(* IEC 61131-3 sources: STVM/tests/functional, 4 files *)

(* ---- io_test.st ---- *)
(*
 * ============================================================================
 * STVM IO 功能综合测试 v3
 * 覆盖: 数字IO / 模拟IO / 安全输出 / 信号缩放 / PID
 * 运行: stvm tests/functional/io_test.st -I
 * ============================================================================
 *)

PROGRAM IOFunctionalTest
VAR_EXTERNAL
    button  AT %IX0.0 : BOOL;
    led     AT %QX0.0 : BOOL;
    adc_raw AT %IW0   : INT;
    pwm_out AT %QW0   : INT;
END_VAR
VAR
    raw_value   : INT;
    scaled_temp : REAL;
    error_flag  : BOOL;
    io_count    : INT;
    setpoint    : REAL;
    process_val : REAL;
    pid_output  : REAL;
    kp          : REAL;
    ki          : REAL;
    kd          : REAL;
    error_val   : REAL;
    integral    : REAL;
    derivative  : REAL;
    last_error  : REAL;
END_VAR

    PRINT('');
    PRINT('========================================');
    PRINT('  STVM IO 功能综合测试');
    PRINT('========================================');

    (* 数字 IO *)
    PRINT('--- 数字 IO ---');
    PRINT('DI button: %d', button);
    led := button;
    PRINT('DO led: %d', led);

    (* 模拟 IO *)
    PRINT('--- 模拟 IO ---');
    PRINT('AI raw: %d', adc_raw);
    pwm_out := 500;
    PRINT('AO pwm: %d', pwm_out);

    (* 信号缩放 *)
    PRINT('--- 缩放 ---');
    raw_value := adc_raw;
    scaled_temp := raw_value * 0.1;
    PRINT('Scaled: %f', scaled_temp);

    (* IO 安全检查 *)
    PRINT('--- 安全 ---');
    error_flag := FALSE;
    IF adc_raw < 0 THEN
        error_flag := TRUE;
    END_IF;
    IF error_flag THEN
        led := FALSE;
        pwm_out := 0;
        PRINT('SAFE: output disabled');
    END_IF;

    (* PID 演示 *)
    PRINT('--- PID ---');
    kp := 1.5;
    ki := 1.0;
    kd := 0.5;
    setpoint := 25.0;
    process_val := scaled_temp;
    error_val := setpoint - process_val;
    integral := integral + error_val * 0.1;
    derivative := (error_val - last_error) / 0.1;
    last_error := error_val;
    pid_output := kp * error_val + ki * integral + kd * derivative;
    PRINT('PID: SP=%f PV=%f OUT=%f', setpoint, process_val, pid_output);

    (* 周期计数器 *)
    io_count := io_count + 1;
    PRINT('IO cycle: %d', io_count);

    PRINT('========================================');
    PRINT('  IO 测试完成');
    PRINT('========================================');
END_PROGRAM

(* ---- reactor_2oo4_test.st ---- *)
(*
 * ============================================================================
 * STVM 极限性能测试 - 核反应堆 2oo4 安全控制系统 [IEC 61508 SIL3]
 * ============================================================================
 *
 * 架构:
 *   - 4 通道冗余传感器 (A/B/C/D)，每组 8 个传感器
 *   - 2oo4 表决逻辑 (4 取 2 触发)
 *   - 多重质量位传播与验证
 *   - PID 控制回路 x4 (温度/压力/流量/水位)
 *   - 安全联锁矩阵 (16x16)
 *   - 启动/运行/停机/紧急状态机
 *   - 报警管理 (16 类报警, 4 级优先级)
 *   - 所有循环带 @LOOP_MAX 标注
 *
 * 规模: ~10000 行 ST 代码, ~500+ 变量, ~80+ 函数
 * ============================================================================
 *)

PROGRAM Reactor2oo4Control

(* ================================================================ *)
(* 全局配置常量 *)
(* ================================================================ *)
VAR
    (* 系统状态 *)
    SYS_IDLE        : INT := 0;
    SYS_STARTUP     : INT := 1;
    SYS_RUNNING     : INT := 2;
    SYS_SHUTDOWN    : INT := 3;
    SYS_EMERGENCY   : INT := 4;
    system_state    : INT := 0;

    (* 安全阈值 *)
    TEMP_TRIP       : REAL := 650.0;
    PRESS_TRIP      : REAL := 15.5;
    FLOW_MIN        : REAL := 100.0;
    LEVEL_MIN       : REAL := 2.0;
    LEVEL_MAX       : REAL := 8.0;

    (* 2oo4 表决配置 *)
    VOTE_THRESHOLD  : INT := 2;
    CHANNEL_FAULT   : INT := -1;
    CHANNEL_OK      : INT := 0;

    (* 全局计数器 *)
    scan_counter    : INT := 0;
    trip_counter    : INT := 0;
    alarm_counter   : INT := 0;
    fault_counter   : INT := 0;

    (* 通用临时变量 *)
    tmp_int         : INT;
    tmp_real        : REAL;
    tmp_bool        : BOOL;
    loop_idx        : INT;
    ch_idx          : INT;
    sn_idx          : INT;
END_VAR

(* ================================================================ *)
(* 通道传感器数据 (4 通道 x 8 传感器/通道 = 32 路) *)
(* ================================================================ *)

(* 通道传感器定义 (32路) *)
FUNCTION ReadChannelA_Sensor0 : QREAL
    ReadChannelA_Sensor0 := MakeQReal(25.0, 0);
END_FUNCTION

FUNCTION ValidateChannelA_Sensor0 : BOOL
VAR_INPUT
    input_val : QREAL;
    min_limit : REAL;
    max_limit : REAL;
END_VAR
    tmp_real := ToReal(input_val);
    tmp_int := GetQuality(input_val);
    tmp_bool := FALSE;
    IF tmp_int = 0 THEN
        IF tmp_real >= min_limit THEN
            IF tmp_real <= max_limit THEN
                tmp_bool := TRUE;
            END_IF;
        END_IF;
    END_IF;
    ValidateChannelA_Sensor0 := tmp_bool;
END_FUNCTION

FUNCTION ReadChannelA_Sensor1 : QREAL
    ReadChannelA_Sensor1 := MakeQReal(25.0, 0);
END_FUNCTION

FUNCTION ValidateChannelA_Sensor1 : BOOL
VAR_INPUT
    input_val : QREAL;
    min_limit : REAL;
    max_limit : REAL;
END_VAR
    tmp_real := ToReal(input_val);
    tmp_int := GetQuality(input_val);
    tmp_bool := FALSE;
    IF tmp_int = 0 THEN
        IF tmp_real >= min_limit THEN
            IF tmp_real <= max_limit THEN
                tmp_bool := TRUE;
            END_IF;
        END_IF;
    END_IF;
    ValidateChannelA_Sensor1 := tmp_bool;
END_FUNCTION

FUNCTION ReadChannelA_Sensor2 : QREAL
    ReadChannelA_Sensor2 := MakeQReal(25.0, 0);
END_FUNCTION

FUNCTION ValidateChannelA_Sensor2 : BOOL
VAR_INPUT
    input_val : QREAL;
    min_limit : REAL;
    max_limit : REAL;
END_VAR
    tmp_real := ToReal(input_val);
    tmp_int := GetQuality(input_val);
    tmp_bool := FALSE;
    IF tmp_int = 0 THEN
        IF tmp_real >= min_limit THEN
            IF tmp_real <= max_limit THEN
                tmp_bool := TRUE;
            END_IF;
        END_IF;
    END_IF;
    ValidateChannelA_Sensor2 := tmp_bool;
END_FUNCTION

FUNCTION ReadChannelA_Sensor3 : QREAL
    ReadChannelA_Sensor3 := MakeQReal(25.0, 0);
END_FUNCTION

FUNCTION ValidateChannelA_Sensor3 : BOOL
VAR_INPUT
    input_val : QREAL;
    min_limit : REAL;
    max_limit : REAL;
END_VAR
    tmp_real := ToReal(input_val);
    tmp_int := GetQuality(input_val);
    tmp_bool := FALSE;
    IF tmp_int = 0 THEN
        IF tmp_real >= min_limit THEN
            IF tmp_real <= max_limit THEN
                tmp_bool := TRUE;
            END_IF;
        END_IF;
    END_IF;
    ValidateChannelA_Sensor3 := tmp_bool;
END_FUNCTION

FUNCTION ReadChannelA_Sensor4 : QREAL
    ReadChannelA_Sensor4 := MakeQReal(25.0, 0);
END_FUNCTION

FUNCTION ValidateChannelA_Sensor4 : BOOL
VAR_INPUT
    input_val : QREAL;
    min_limit : REAL;
    max_limit : REAL;
END_VAR
    tmp_real := ToReal(input_val);
    tmp_int := GetQuality(input_val);
    tmp_bool := FALSE;
    IF tmp_int = 0 THEN
        IF tmp_real >= min_limit THEN
            IF tmp_real <= max_limit THEN
                tmp_bool := TRUE;
            END_IF;
        END_IF;
    END_IF;
    ValidateChannelA_Sensor4 := tmp_bool;
END_FUNCTION

FUNCTION ReadChannelA_Sensor5 : QREAL
    ReadChannelA_Sensor5 := MakeQReal(25.0, 0);
END_FUNCTION

FUNCTION ValidateChannelA_Sensor5 : BOOL
VAR_INPUT
    input_val : QREAL;
    min_limit : REAL;
    max_limit : REAL;
END_VAR
    tmp_real := ToReal(input_val);
    tmp_int := GetQuality(input_val);
    tmp_bool := FALSE;
    IF tmp_int = 0 THEN
        IF tmp_real >= min_limit THEN
            IF tmp_real <= max_limit THEN
                tmp_bool := TRUE;
            END_IF;
        END_IF;
    END_IF;
    ValidateChannelA_Sensor5 := tmp_bool;
END_FUNCTION

FUNCTION ReadChannelA_Sensor6 : QREAL
    ReadChannelA_Sensor6 := MakeQReal(25.0, 0);
END_FUNCTION

FUNCTION ValidateChannelA_Sensor6 : BOOL
VAR_INPUT
    input_val : QREAL;
    min_limit : REAL;
    max_limit : REAL;
END_VAR
    tmp_real := ToReal(input_val);
    tmp_int := GetQuality(input_val);
    tmp_bool := FALSE;
    IF tmp_int = 0 THEN
        IF tmp_real >= min_limit THEN
            IF tmp_real <= max_limit THEN
                tmp_bool := TRUE;
            END_IF;
        END_IF;
    END_IF;
    ValidateChannelA_Sensor6 := tmp_bool;
END_FUNCTION

FUNCTION ReadChannelA_Sensor7 : QREAL
    ReadChannelA_Sensor7 := MakeQReal(25.0, 0);
END_FUNCTION

FUNCTION ValidateChannelA_Sensor7 : BOOL
VAR_INPUT
    input_val : QREAL;
    min_limit : REAL;
    max_limit : REAL;
END_VAR
    tmp_real := ToReal(input_val);
    tmp_int := GetQuality(input_val);
    tmp_bool := FALSE;
    IF tmp_int = 0 THEN
        IF tmp_real >= min_limit THEN
            IF tmp_real <= max_limit THEN
                tmp_bool := TRUE;
            END_IF;
        END_IF;
    END_IF;
    ValidateChannelA_Sensor7 := tmp_bool;
END_FUNCTION

FUNCTION ReadChannelB_Sensor0 : QREAL
    ReadChannelB_Sensor0 := MakeQReal(25.0, 0);
END_FUNCTION

FUNCTION ValidateChannelB_Sensor0 : BOOL
VAR_INPUT
    input_val : QREAL;
    min_limit : REAL;
    max_limit : REAL;
END_VAR
    tmp_real := ToReal(input_val);
    tmp_int := GetQuality(input_val);
    tmp_bool := FALSE;
    IF tmp_int = 0 THEN
        IF tmp_real >= min_limit THEN
            IF tmp_real <= max_limit THEN
                tmp_bool := TRUE;
            END_IF;
        END_IF;
    END_IF;
    ValidateChannelB_Sensor0 := tmp_bool;
END_FUNCTION

FUNCTION ReadChannelB_Sensor1 : QREAL
    ReadChannelB_Sensor1 := MakeQReal(25.0, 0);
END_FUNCTION

FUNCTION ValidateChannelB_Sensor1 : BOOL
VAR_INPUT
    input_val : QREAL;
    min_limit : REAL;
    max_limit : REAL;
END_VAR
    tmp_real := ToReal(input_val);
    tmp_int := GetQuality(input_val);
    tmp_bool := FALSE;
    IF tmp_int = 0 THEN
        IF tmp_real >= min_limit THEN
            IF tmp_real <= max_limit THEN
                tmp_bool := TRUE;
            END_IF;
        END_IF;
    END_IF;
    ValidateChannelB_Sensor1 := tmp_bool;
END_FUNCTION

FUNCTION ReadChannelB_Sensor2 : QREAL
    ReadChannelB_Sensor2 := MakeQReal(25.0, 0);
END_FUNCTION

FUNCTION ValidateChannelB_Sensor2 : BOOL
VAR_INPUT
    input_val : QREAL;
    min_limit : REAL;
    max_limit : REAL;
END_VAR
    tmp_real := ToReal(input_val);
    tmp_int := GetQuality(input_val);
    tmp_bool := FALSE;
    IF tmp_int = 0 THEN
        IF tmp_real >= min_limit THEN
            IF tmp_real <= max_limit THEN
                tmp_bool := TRUE;
            END_IF;
        END_IF;
    END_IF;
    ValidateChannelB_Sensor2 := tmp_bool;
END_FUNCTION

FUNCTION ReadChannelB_Sensor3 : QREAL
    ReadChannelB_Sensor3 := MakeQReal(25.0, 0);
END_FUNCTION

FUNCTION ValidateChannelB_Sensor3 : BOOL
VAR_INPUT
    input_val : QREAL;
    min_limit : REAL;
    max_limit : REAL;
END_VAR
    tmp_real := ToReal(input_val);
    tmp_int := GetQuality(input_val);
    tmp_bool := FALSE;
    IF tmp_int = 0 THEN
        IF tmp_real >= min_limit THEN
            IF tmp_real <= max_limit THEN
                tmp_bool := TRUE;
            END_IF;
        END_IF;
    END_IF;
    ValidateChannelB_Sensor3 := tmp_bool;
END_FUNCTION

FUNCTION ReadChannelB_Sensor4 : QREAL
    ReadChannelB_Sensor4 := MakeQReal(25.0, 0);
END_FUNCTION

FUNCTION ValidateChannelB_Sensor4 : BOOL
VAR_INPUT
    input_val : QREAL;
    min_limit : REAL;
    max_limit : REAL;
END_VAR
    tmp_real := ToReal(input_val);
    tmp_int := GetQuality(input_val);
    tmp_bool := FALSE;
    IF tmp_int = 0 THEN
        IF tmp_real >= min_limit THEN
            IF tmp_real <= max_limit THEN
                tmp_bool := TRUE;
            END_IF;
        END_IF;
    END_IF;
    ValidateChannelB_Sensor4 := tmp_bool;
END_FUNCTION

FUNCTION ReadChannelB_Sensor5 : QREAL
    ReadChannelB_Sensor5 := MakeQReal(25.0, 0);
END_FUNCTION

FUNCTION ValidateChannelB_Sensor5 : BOOL
VAR_INPUT
    input_val : QREAL;
    min_limit : REAL;
    max_limit : REAL;
END_VAR
    tmp_real := ToReal(input_val);
    tmp_int := GetQuality(input_val);
    tmp_bool := FALSE;
    IF tmp_int = 0 THEN
        IF tmp_real >= min_limit THEN
            IF tmp_real <= max_limit THEN
                tmp_bool := TRUE;
            END_IF;
        END_IF;
    END_IF;
    ValidateChannelB_Sensor5 := tmp_bool;
END_FUNCTION

FUNCTION ReadChannelB_Sensor6 : QREAL
    ReadChannelB_Sensor6 := MakeQReal(25.0, 0);
END_FUNCTION

FUNCTION ValidateChannelB_Sensor6 : BOOL
VAR_INPUT
    input_val : QREAL;
    min_limit : REAL;
    max_limit : REAL;
END_VAR
    tmp_real := ToReal(input_val);
    tmp_int := GetQuality(input_val);
    tmp_bool := FALSE;
    IF tmp_int = 0 THEN
        IF tmp_real >= min_limit THEN
            IF tmp_real <= max_limit THEN
                tmp_bool := TRUE;
            END_IF;
        END_IF;
    END_IF;
    ValidateChannelB_Sensor6 := tmp_bool;
END_FUNCTION

FUNCTION ReadChannelB_Sensor7 : QREAL
    ReadChannelB_Sensor7 := MakeQReal(25.0, 0);
END_FUNCTION

FUNCTION ValidateChannelB_Sensor7 : BOOL
VAR_INPUT
    input_val : QREAL;
    min_limit : REAL;
    max_limit : REAL;
END_VAR
    tmp_real := ToReal(input_val);
    tmp_int := GetQuality(input_val);
    tmp_bool := FALSE;
    IF tmp_int = 0 THEN
        IF tmp_real >= min_limit THEN
            IF tmp_real <= max_limit THEN
                tmp_bool := TRUE;
            END_IF;
        END_IF;
    END_IF;
    ValidateChannelB_Sensor7 := tmp_bool;
END_FUNCTION

FUNCTION ReadChannelC_Sensor0 : QREAL
    ReadChannelC_Sensor0 := MakeQReal(25.0, 0);
END_FUNCTION

FUNCTION ValidateChannelC_Sensor0 : BOOL
VAR_INPUT
    input_val : QREAL;
    min_limit : REAL;
    max_limit : REAL;
END_VAR
    tmp_real := ToReal(input_val);
    tmp_int := GetQuality(input_val);
    tmp_bool := FALSE;
    IF tmp_int = 0 THEN
        IF tmp_real >= min_limit THEN
            IF tmp_real <= max_limit THEN
                tmp_bool := TRUE;
            END_IF;
        END_IF;
    END_IF;
    ValidateChannelC_Sensor0 := tmp_bool;
END_FUNCTION

FUNCTION ReadChannelC_Sensor1 : QREAL
    ReadChannelC_Sensor1 := MakeQReal(25.0, 0);
END_FUNCTION

FUNCTION ValidateChannelC_Sensor1 : BOOL
VAR_INPUT
    input_val : QREAL;
    min_limit : REAL;
    max_limit : REAL;
END_VAR
    tmp_real := ToReal(input_val);
    tmp_int := GetQuality(input_val);
    tmp_bool := FALSE;
    IF tmp_int = 0 THEN
        IF tmp_real >= min_limit THEN
            IF tmp_real <= max_limit THEN
                tmp_bool := TRUE;
            END_IF;
        END_IF;
    END_IF;
    ValidateChannelC_Sensor1 := tmp_bool;
END_FUNCTION

FUNCTION ReadChannelC_Sensor2 : QREAL
    ReadChannelC_Sensor2 := MakeQReal(25.0, 0);
END_FUNCTION

FUNCTION ValidateChannelC_Sensor2 : BOOL
VAR_INPUT
    input_val : QREAL;
    min_limit : REAL;
    max_limit : REAL;
END_VAR
    tmp_real := ToReal(input_val);
    tmp_int := GetQuality(input_val);
    tmp_bool := FALSE;
    IF tmp_int = 0 THEN
        IF tmp_real >= min_limit THEN
            IF tmp_real <= max_limit THEN
                tmp_bool := TRUE;
            END_IF;
        END_IF;
    END_IF;
    ValidateChannelC_Sensor2 := tmp_bool;
END_FUNCTION

FUNCTION ReadChannelC_Sensor3 : QREAL
    ReadChannelC_Sensor3 := MakeQReal(25.0, 0);
END_FUNCTION

FUNCTION ValidateChannelC_Sensor3 : BOOL
VAR_INPUT
    input_val : QREAL;
    min_limit : REAL;
    max_limit : REAL;
END_VAR
    tmp_real := ToReal(input_val);
    tmp_int := GetQuality(input_val);
    tmp_bool := FALSE;
    IF tmp_int = 0 THEN
        IF tmp_real >= min_limit THEN
            IF tmp_real <= max_limit THEN
                tmp_bool := TRUE;
            END_IF;
        END_IF;
    END_IF;
    ValidateChannelC_Sensor3 := tmp_bool;
END_FUNCTION

FUNCTION ReadChannelC_Sensor4 : QREAL
    ReadChannelC_Sensor4 := MakeQReal(25.0, 0);
END_FUNCTION

FUNCTION ValidateChannelC_Sensor4 : BOOL
VAR_INPUT
    input_val : QREAL;
    min_limit : REAL;
    max_limit : REAL;
END_VAR
    tmp_real := ToReal(input_val);
    tmp_int := GetQuality(input_val);
    tmp_bool := FALSE;
    IF tmp_int = 0 THEN
        IF tmp_real >= min_limit THEN
            IF tmp_real <= max_limit THEN
                tmp_bool := TRUE;
            END_IF;
        END_IF;
    END_IF;
    ValidateChannelC_Sensor4 := tmp_bool;
END_FUNCTION

FUNCTION ReadChannelC_Sensor5 : QREAL
    ReadChannelC_Sensor5 := MakeQReal(25.0, 0);
END_FUNCTION

FUNCTION ValidateChannelC_Sensor5 : BOOL
VAR_INPUT
    input_val : QREAL;
    min_limit : REAL;
    max_limit : REAL;
END_VAR
    tmp_real := ToReal(input_val);
    tmp_int := GetQuality(input_val);
    tmp_bool := FALSE;
    IF tmp_int = 0 THEN
        IF tmp_real >= min_limit THEN
            IF tmp_real <= max_limit THEN
                tmp_bool := TRUE;
            END_IF;
        END_IF;
    END_IF;
    ValidateChannelC_Sensor5 := tmp_bool;
END_FUNCTION

FUNCTION ReadChannelC_Sensor6 : QREAL
    ReadChannelC_Sensor6 := MakeQReal(25.0, 0);
END_FUNCTION

FUNCTION ValidateChannelC_Sensor6 : BOOL
VAR_INPUT
    input_val : QREAL;
    min_limit : REAL;
    max_limit : REAL;
END_VAR
    tmp_real := ToReal(input_val);
    tmp_int := GetQuality(input_val);
    tmp_bool := FALSE;
    IF tmp_int = 0 THEN
        IF tmp_real >= min_limit THEN
            IF tmp_real <= max_limit THEN
                tmp_bool := TRUE;
            END_IF;
        END_IF;
    END_IF;
    ValidateChannelC_Sensor6 := tmp_bool;
END_FUNCTION

FUNCTION ReadChannelC_Sensor7 : QREAL
    ReadChannelC_Sensor7 := MakeQReal(25.0, 0);
END_FUNCTION

FUNCTION ValidateChannelC_Sensor7 : BOOL
VAR_INPUT
    input_val : QREAL;
    min_limit : REAL;
    max_limit : REAL;
END_VAR
    tmp_real := ToReal(input_val);
    tmp_int := GetQuality(input_val);
    tmp_bool := FALSE;
    IF tmp_int = 0 THEN
        IF tmp_real >= min_limit THEN
            IF tmp_real <= max_limit THEN
                tmp_bool := TRUE;
            END_IF;
        END_IF;
    END_IF;
    ValidateChannelC_Sensor7 := tmp_bool;
END_FUNCTION

FUNCTION ReadChannelD_Sensor0 : QREAL
    ReadChannelD_Sensor0 := MakeQReal(25.0, 0);
END_FUNCTION

FUNCTION ValidateChannelD_Sensor0 : BOOL
VAR_INPUT
    input_val : QREAL;
    min_limit : REAL;
    max_limit : REAL;
END_VAR
    tmp_real := ToReal(input_val);
    tmp_int := GetQuality(input_val);
    tmp_bool := FALSE;
    IF tmp_int = 0 THEN
        IF tmp_real >= min_limit THEN
            IF tmp_real <= max_limit THEN
                tmp_bool := TRUE;
            END_IF;
        END_IF;
    END_IF;
    ValidateChannelD_Sensor0 := tmp_bool;
END_FUNCTION

FUNCTION ReadChannelD_Sensor1 : QREAL
    ReadChannelD_Sensor1 := MakeQReal(25.0, 0);
END_FUNCTION

FUNCTION ValidateChannelD_Sensor1 : BOOL
VAR_INPUT
    input_val : QREAL;
    min_limit : REAL;
    max_limit : REAL;
END_VAR
    tmp_real := ToReal(input_val);
    tmp_int := GetQuality(input_val);
    tmp_bool := FALSE;
    IF tmp_int = 0 THEN
        IF tmp_real >= min_limit THEN
            IF tmp_real <= max_limit THEN
                tmp_bool := TRUE;
            END_IF;
        END_IF;
    END_IF;
    ValidateChannelD_Sensor1 := tmp_bool;
END_FUNCTION

FUNCTION ReadChannelD_Sensor2 : QREAL
    ReadChannelD_Sensor2 := MakeQReal(25.0, 0);
END_FUNCTION

FUNCTION ValidateChannelD_Sensor2 : BOOL
VAR_INPUT
    input_val : QREAL;
    min_limit : REAL;
    max_limit : REAL;
END_VAR
    tmp_real := ToReal(input_val);
    tmp_int := GetQuality(input_val);
    tmp_bool := FALSE;
    IF tmp_int = 0 THEN
        IF tmp_real >= min_limit THEN
            IF tmp_real <= max_limit THEN
                tmp_bool := TRUE;
            END_IF;
        END_IF;
    END_IF;
    ValidateChannelD_Sensor2 := tmp_bool;
END_FUNCTION

FUNCTION ReadChannelD_Sensor3 : QREAL
    ReadChannelD_Sensor3 := MakeQReal(25.0, 0);
END_FUNCTION

FUNCTION ValidateChannelD_Sensor3 : BOOL
VAR_INPUT
    input_val : QREAL;
    min_limit : REAL;
    max_limit : REAL;
END_VAR
    tmp_real := ToReal(input_val);
    tmp_int := GetQuality(input_val);
    tmp_bool := FALSE;
    IF tmp_int = 0 THEN
        IF tmp_real >= min_limit THEN
            IF tmp_real <= max_limit THEN
                tmp_bool := TRUE;
            END_IF;
        END_IF;
    END_IF;
    ValidateChannelD_Sensor3 := tmp_bool;
END_FUNCTION

FUNCTION ReadChannelD_Sensor4 : QREAL
    ReadChannelD_Sensor4 := MakeQReal(25.0, 0);
END_FUNCTION

FUNCTION ValidateChannelD_Sensor4 : BOOL
VAR_INPUT
    input_val : QREAL;
    min_limit : REAL;
    max_limit : REAL;
END_VAR
    tmp_real := ToReal(input_val);
    tmp_int := GetQuality(input_val);
    tmp_bool := FALSE;
    IF tmp_int = 0 THEN
        IF tmp_real >= min_limit THEN
            IF tmp_real <= max_limit THEN
                tmp_bool := TRUE;
            END_IF;
        END_IF;
    END_IF;
    ValidateChannelD_Sensor4 := tmp_bool;
END_FUNCTION

FUNCTION ReadChannelD_Sensor5 : QREAL
    ReadChannelD_Sensor5 := MakeQReal(25.0, 0);
END_FUNCTION

FUNCTION ValidateChannelD_Sensor5 : BOOL
VAR_INPUT
    input_val : QREAL;
    min_limit : REAL;
    max_limit : REAL;
END_VAR
    tmp_real := ToReal(input_val);
    tmp_int := GetQuality(input_val);
    tmp_bool := FALSE;
    IF tmp_int = 0 THEN
        IF tmp_real >= min_limit THEN
            IF tmp_real <= max_limit THEN
                tmp_bool := TRUE;
            END_IF;
        END_IF;
    END_IF;
    ValidateChannelD_Sensor5 := tmp_bool;
END_FUNCTION

FUNCTION ReadChannelD_Sensor6 : QREAL
    ReadChannelD_Sensor6 := MakeQReal(25.0, 0);
END_FUNCTION

FUNCTION ValidateChannelD_Sensor6 : BOOL
VAR_INPUT
    input_val : QREAL;
    min_limit : REAL;
    max_limit : REAL;
END_VAR
    tmp_real := ToReal(input_val);
    tmp_int := GetQuality(input_val);
    tmp_bool := FALSE;
    IF tmp_int = 0 THEN
        IF tmp_real >= min_limit THEN
            IF tmp_real <= max_limit THEN
                tmp_bool := TRUE;
            END_IF;
        END_IF;
    END_IF;
    ValidateChannelD_Sensor6 := tmp_bool;
END_FUNCTION

FUNCTION ReadChannelD_Sensor7 : QREAL
    ReadChannelD_Sensor7 := MakeQReal(25.0, 0);
END_FUNCTION

FUNCTION ValidateChannelD_Sensor7 : BOOL
VAR_INPUT
    input_val : QREAL;
    min_limit : REAL;
    max_limit : REAL;
END_VAR
    tmp_real := ToReal(input_val);
    tmp_int := GetQuality(input_val);
    tmp_bool := FALSE;
    IF tmp_int = 0 THEN
        IF tmp_real >= min_limit THEN
            IF tmp_real <= max_limit THEN
                tmp_bool := TRUE;
            END_IF;
        END_IF;
    END_IF;
    ValidateChannelD_Sensor7 := tmp_bool;
END_FUNCTION

(* ================================================================ *)
(* 2oo4 表决逻辑 *)
(* ================================================================ *)

FUNCTION Vote2oo4_Bool : BOOL
VAR_INPUT
    ch_a : BOOL;
    ch_b : BOOL;
    ch_c : BOOL;
    ch_d : BOOL;
END_VAR
    tmp_int := 0;
    IF ch_a THEN tmp_int := tmp_int + 1; END_IF;
    IF ch_b THEN tmp_int := tmp_int + 1; END_IF;
    IF ch_c THEN tmp_int := tmp_int + 1; END_IF;
    IF ch_d THEN tmp_int := tmp_int + 1; END_IF;
    Vote2oo4_Bool := (tmp_int >= VOTE_THRESHOLD);
END_FUNCTION

FUNCTION Vote2oo4_Real : REAL
VAR_INPUT
    ch_a : REAL;
    ch_b : REAL;
    ch_c : REAL;
    ch_d : REAL;
END_VAR
    tmp_real := ch_a + ch_b + ch_c + ch_d;
    Vote2oo4_Real := tmp_real / 4.0;
END_FUNCTION

FUNCTION Vote2oo4_QReal : QREAL
VAR_INPUT
    ch_a : QREAL;
    ch_b : QREAL;
    ch_c : QREAL;
    ch_d : QREAL;
END_VAR
    tmp_real := ToReal(ch_a) + ToReal(ch_b) + ToReal(ch_c) + ToReal(ch_d);
    Vote2oo4_QReal := MakeQReal(tmp_real / 4.0, 0);
END_FUNCTION

(* ================================================================ *)
(* @LOOP_MAX(10000) - 传感器组 0 2oo4 表决 *)
(* ================================================================ *)
FUNCTION SensorGroup0_Vote : QREAL
VAR
    s_a : QREAL;
    s_b : QREAL;
    s_c : QREAL;
    s_d : QREAL;
    v_a : BOOL;
    v_b : BOOL;
    v_c : BOOL;
    v_d : BOOL;
    vt : BOOL;
    result : QREAL;
END_VAR
    s_a := ReadChannelA_Sensor0();
    s_b := ReadChannelB_Sensor0();
    s_c := ReadChannelC_Sensor0();
    s_d := ReadChannelD_Sensor0();

    v_a := ValidateChannelA_Sensor0(s_a, 0.0, 1000.0);
    v_b := ValidateChannelB_Sensor0(s_b, 0.0, 1000.0);
    v_c := ValidateChannelC_Sensor0(s_c, 0.0, 1000.0);
    v_d := ValidateChannelD_Sensor0(s_d, 0.0, 1000.0);

    vt := Vote2oo4_Bool(v_a, v_b, v_c, v_d);
    IF vt THEN
        result := Vote2oo4_QReal(s_a, s_b, s_c, s_d);
    ELSE
        result := MakeQReal(0.0, 3);
    END_IF;
    SensorGroup0_Vote := result;
END_FUNCTION

(* ================================================================ *)
(* @LOOP_MAX(10000) - 传感器组 1 2oo4 表决 *)
(* ================================================================ *)
FUNCTION SensorGroup1_Vote : QREAL
VAR
    s_a : QREAL;
    s_b : QREAL;
    s_c : QREAL;
    s_d : QREAL;
    v_a : BOOL;
    v_b : BOOL;
    v_c : BOOL;
    v_d : BOOL;
    vt : BOOL;
    result : QREAL;
END_VAR
    s_a := ReadChannelA_Sensor1();
    s_b := ReadChannelB_Sensor1();
    s_c := ReadChannelC_Sensor1();
    s_d := ReadChannelD_Sensor1();

    v_a := ValidateChannelA_Sensor1(s_a, 0.0, 1000.0);
    v_b := ValidateChannelB_Sensor1(s_b, 0.0, 1000.0);
    v_c := ValidateChannelC_Sensor1(s_c, 0.0, 1000.0);
    v_d := ValidateChannelD_Sensor1(s_d, 0.0, 1000.0);

    vt := Vote2oo4_Bool(v_a, v_b, v_c, v_d);
    IF vt THEN
        result := Vote2oo4_QReal(s_a, s_b, s_c, s_d);
    ELSE
        result := MakeQReal(0.0, 3);
    END_IF;
    SensorGroup1_Vote := result;
END_FUNCTION

(* ================================================================ *)
(* @LOOP_MAX(10000) - 传感器组 2 2oo4 表决 *)
(* ================================================================ *)
FUNCTION SensorGroup2_Vote : QREAL
VAR
    s_a : QREAL;
    s_b : QREAL;
    s_c : QREAL;
    s_d : QREAL;
    v_a : BOOL;
    v_b : BOOL;
    v_c : BOOL;
    v_d : BOOL;
    vt : BOOL;
    result : QREAL;
END_VAR
    s_a := ReadChannelA_Sensor2();
    s_b := ReadChannelB_Sensor2();
    s_c := ReadChannelC_Sensor2();
    s_d := ReadChannelD_Sensor2();

    v_a := ValidateChannelA_Sensor2(s_a, 0.0, 1000.0);
    v_b := ValidateChannelB_Sensor2(s_b, 0.0, 1000.0);
    v_c := ValidateChannelC_Sensor2(s_c, 0.0, 1000.0);
    v_d := ValidateChannelD_Sensor2(s_d, 0.0, 1000.0);

    vt := Vote2oo4_Bool(v_a, v_b, v_c, v_d);
    IF vt THEN
        result := Vote2oo4_QReal(s_a, s_b, s_c, s_d);
    ELSE
        result := MakeQReal(0.0, 3);
    END_IF;
    SensorGroup2_Vote := result;
END_FUNCTION

(* ================================================================ *)
(* @LOOP_MAX(10000) - 传感器组 3 2oo4 表决 *)
(* ================================================================ *)
FUNCTION SensorGroup3_Vote : QREAL
VAR
    s_a : QREAL;
    s_b : QREAL;
    s_c : QREAL;
    s_d : QREAL;
    v_a : BOOL;
    v_b : BOOL;
    v_c : BOOL;
    v_d : BOOL;
    vt : BOOL;
    result : QREAL;
END_VAR
    s_a := ReadChannelA_Sensor3();
    s_b := ReadChannelB_Sensor3();
    s_c := ReadChannelC_Sensor3();
    s_d := ReadChannelD_Sensor3();

    v_a := ValidateChannelA_Sensor3(s_a, 0.0, 1000.0);
    v_b := ValidateChannelB_Sensor3(s_b, 0.0, 1000.0);
    v_c := ValidateChannelC_Sensor3(s_c, 0.0, 1000.0);
    v_d := ValidateChannelD_Sensor3(s_d, 0.0, 1000.0);

    vt := Vote2oo4_Bool(v_a, v_b, v_c, v_d);
    IF vt THEN
        result := Vote2oo4_QReal(s_a, s_b, s_c, s_d);
    ELSE
        result := MakeQReal(0.0, 3);
    END_IF;
    SensorGroup3_Vote := result;
END_FUNCTION

(* ================================================================ *)
(* @LOOP_MAX(10000) - 传感器组 4 2oo4 表决 *)
(* ================================================================ *)
FUNCTION SensorGroup4_Vote : QREAL
VAR
    s_a : QREAL;
    s_b : QREAL;
    s_c : QREAL;
    s_d : QREAL;
    v_a : BOOL;
    v_b : BOOL;
    v_c : BOOL;
    v_d : BOOL;
    vt : BOOL;
    result : QREAL;
END_VAR
    s_a := ReadChannelA_Sensor4();
    s_b := ReadChannelB_Sensor4();
    s_c := ReadChannelC_Sensor4();
    s_d := ReadChannelD_Sensor4();

    v_a := ValidateChannelA_Sensor4(s_a, 0.0, 1000.0);
    v_b := ValidateChannelB_Sensor4(s_b, 0.0, 1000.0);
    v_c := ValidateChannelC_Sensor4(s_c, 0.0, 1000.0);
    v_d := ValidateChannelD_Sensor4(s_d, 0.0, 1000.0);

    vt := Vote2oo4_Bool(v_a, v_b, v_c, v_d);
    IF vt THEN
        result := Vote2oo4_QReal(s_a, s_b, s_c, s_d);
    ELSE
        result := MakeQReal(0.0, 3);
    END_IF;
    SensorGroup4_Vote := result;
END_FUNCTION

(* ================================================================ *)
(* @LOOP_MAX(10000) - 传感器组 5 2oo4 表决 *)
(* ================================================================ *)
FUNCTION SensorGroup5_Vote : QREAL
VAR
    s_a : QREAL;
    s_b : QREAL;
    s_c : QREAL;
    s_d : QREAL;
    v_a : BOOL;
    v_b : BOOL;
    v_c : BOOL;
    v_d : BOOL;
    vt : BOOL;
    result : QREAL;
END_VAR
    s_a := ReadChannelA_Sensor5();
    s_b := ReadChannelB_Sensor5();
    s_c := ReadChannelC_Sensor5();
    s_d := ReadChannelD_Sensor5();

    v_a := ValidateChannelA_Sensor5(s_a, 0.0, 1000.0);
    v_b := ValidateChannelB_Sensor5(s_b, 0.0, 1000.0);
    v_c := ValidateChannelC_Sensor5(s_c, 0.0, 1000.0);
    v_d := ValidateChannelD_Sensor5(s_d, 0.0, 1000.0);

    vt := Vote2oo4_Bool(v_a, v_b, v_c, v_d);
    IF vt THEN
        result := Vote2oo4_QReal(s_a, s_b, s_c, s_d);
    ELSE
        result := MakeQReal(0.0, 3);
    END_IF;
    SensorGroup5_Vote := result;
END_FUNCTION

(* ================================================================ *)
(* @LOOP_MAX(10000) - 传感器组 6 2oo4 表决 *)
(* ================================================================ *)
FUNCTION SensorGroup6_Vote : QREAL
VAR
    s_a : QREAL;
    s_b : QREAL;
    s_c : QREAL;
    s_d : QREAL;
    v_a : BOOL;
    v_b : BOOL;
    v_c : BOOL;
    v_d : BOOL;
    vt : BOOL;
    result : QREAL;
END_VAR
    s_a := ReadChannelA_Sensor6();
    s_b := ReadChannelB_Sensor6();
    s_c := ReadChannelC_Sensor6();
    s_d := ReadChannelD_Sensor6();

    v_a := ValidateChannelA_Sensor6(s_a, 0.0, 1000.0);
    v_b := ValidateChannelB_Sensor6(s_b, 0.0, 1000.0);
    v_c := ValidateChannelC_Sensor6(s_c, 0.0, 1000.0);
    v_d := ValidateChannelD_Sensor6(s_d, 0.0, 1000.0);

    vt := Vote2oo4_Bool(v_a, v_b, v_c, v_d);
    IF vt THEN
        result := Vote2oo4_QReal(s_a, s_b, s_c, s_d);
    ELSE
        result := MakeQReal(0.0, 3);
    END_IF;
    SensorGroup6_Vote := result;
END_FUNCTION

(* ================================================================ *)
(* @LOOP_MAX(10000) - 传感器组 7 2oo4 表决 *)
(* ================================================================ *)
FUNCTION SensorGroup7_Vote : QREAL
VAR
    s_a : QREAL;
    s_b : QREAL;
    s_c : QREAL;
    s_d : QREAL;
    v_a : BOOL;
    v_b : BOOL;
    v_c : BOOL;
    v_d : BOOL;
    vt : BOOL;
    result : QREAL;
END_VAR
    s_a := ReadChannelA_Sensor7();
    s_b := ReadChannelB_Sensor7();
    s_c := ReadChannelC_Sensor7();
    s_d := ReadChannelD_Sensor7();

    v_a := ValidateChannelA_Sensor7(s_a, 0.0, 1000.0);
    v_b := ValidateChannelB_Sensor7(s_b, 0.0, 1000.0);
    v_c := ValidateChannelC_Sensor7(s_c, 0.0, 1000.0);
    v_d := ValidateChannelD_Sensor7(s_d, 0.0, 1000.0);

    vt := Vote2oo4_Bool(v_a, v_b, v_c, v_d);
    IF vt THEN
        result := Vote2oo4_QReal(s_a, s_b, s_c, s_d);
    ELSE
        result := MakeQReal(0.0, 3);
    END_IF;
    SensorGroup7_Vote := result;
END_FUNCTION

(* ================================================================ *)
(* PID 控制器 x4 *)
(* ================================================================ *)

FUNCTION PID_Temperature : REAL
VAR_INPUT
    sp : REAL;
    pv : REAL;
END_VAR
VAR
    kp_temp : REAL := 2.5;
    ki_temp : REAL := 0.8;
    kd_temp : REAL := 0.3;
    err     : REAL;
    integ   : REAL;
    deriv   : REAL;
    prev_err: REAL;
END_VAR
    err := sp - pv;
    integ := integ + err * 0.1;
    deriv := (err - prev_err) / 0.1;
    prev_err := err;
    PID_Temperature := kp_temp * err + ki_temp * integ + kd_temp * deriv;
END_FUNCTION

FUNCTION PID_Pressure : REAL
VAR_INPUT
    sp : REAL;
    pv : REAL;
END_VAR
VAR
    kp_val : REAL := 3.0;
    ki_val : REAL := 1.2;
    kd_val : REAL := 0.5;
    err     : REAL;
    integ   : REAL;
    deriv   : REAL;
    prev_err: REAL;
END_VAR
    err := sp - pv;
    integ := integ + err * 0.1;
    deriv := (err - prev_err) / 0.1;
    prev_err := err;
    PID_Pressure := kp_val * err + ki_val * integ + kd_val * deriv;
END_FUNCTION
FUNCTION PID_Flow : REAL
VAR_INPUT
    sp : REAL;
    pv : REAL;
END_VAR
VAR
    kp_val : REAL := 1.5;
    ki_val : REAL := 0.6;
    kd_val : REAL := 0.2;
    err     : REAL;
    integ   : REAL;
    deriv   : REAL;
    prev_err: REAL;
END_VAR
    err := sp - pv;
    integ := integ + err * 0.1;
    deriv := (err - prev_err) / 0.1;
    prev_err := err;
    PID_Flow := kp_val * err + ki_val * integ + kd_val * deriv;
END_FUNCTION
FUNCTION PID_Level : REAL
VAR_INPUT
    sp : REAL;
    pv : REAL;
END_VAR
VAR
    kp_val : REAL := 2.0;
    ki_val : REAL := 0.3;
    kd_val : REAL := 0.1;
    err     : REAL;
    integ   : REAL;
    deriv   : REAL;
    prev_err: REAL;
END_VAR
    err := sp - pv;
    integ := integ + err * 0.1;
    deriv := (err - prev_err) / 0.1;
    prev_err := err;
    PID_Level := kp_val * err + ki_val * integ + kd_val * deriv;
END_FUNCTION
(* ================================================================ *)
(* 安全联锁矩阵 16x16 *)
(* ================================================================ *)

FUNCTION InterlockMatrix : BOOL
VAR_INPUT
    signals : ARRAY[16] OF BOOL;
END_VAR
VAR
    row : INT;
    col : INT;
    result : BOOL;
END_VAR
    result := FALSE;
    FOR row := 0 TO 15 DO
        FOR col := 0 TO 15 DO
            IF signals[row] THEN
                IF signals[col] THEN
                    result := TRUE;
                END_IF;
            END_IF;
        END_FOR;
    END_FOR;
    InterlockMatrix := result;
END_FUNCTION

(* 联锁信号赋值函数 *)
FUNCTION Interlock_R0 : BOOL
VAR_INPUT
    signals : ARRAY[16] OF BOOL;
END_VAR
    Interlock_R0 := signals[0] AND signals[0];
END_FUNCTION
FUNCTION Interlock_R1 : BOOL
VAR_INPUT
    signals : ARRAY[16] OF BOOL;
END_VAR
    Interlock_R1 := signals[1] AND signals[0];
END_FUNCTION
FUNCTION Interlock_R2 : BOOL
VAR_INPUT
    signals : ARRAY[16] OF BOOL;
END_VAR
    Interlock_R2 := signals[2] AND signals[0];
END_FUNCTION
FUNCTION Interlock_R3 : BOOL
VAR_INPUT
    signals : ARRAY[16] OF BOOL;
END_VAR
    Interlock_R3 := signals[3] AND signals[0];
END_FUNCTION
FUNCTION Interlock_R4 : BOOL
VAR_INPUT
    signals : ARRAY[16] OF BOOL;
END_VAR
    Interlock_R4 := signals[4] AND signals[0];
END_FUNCTION
FUNCTION Interlock_R5 : BOOL
VAR_INPUT
    signals : ARRAY[16] OF BOOL;
END_VAR
    Interlock_R5 := signals[5] AND signals[0];
END_FUNCTION
FUNCTION Interlock_R6 : BOOL
VAR_INPUT
    signals : ARRAY[16] OF BOOL;
END_VAR
    Interlock_R6 := signals[6] AND signals[0];
END_FUNCTION
FUNCTION Interlock_R7 : BOOL
VAR_INPUT
    signals : ARRAY[16] OF BOOL;
END_VAR
    Interlock_R7 := signals[7] AND signals[0];
END_FUNCTION
FUNCTION Interlock_R8 : BOOL
VAR_INPUT
    signals : ARRAY[16] OF BOOL;
END_VAR
    Interlock_R8 := signals[8] AND signals[0];
END_FUNCTION
FUNCTION Interlock_R9 : BOOL
VAR_INPUT
    signals : ARRAY[16] OF BOOL;
END_VAR
    Interlock_R9 := signals[9] AND signals[0];
END_FUNCTION
FUNCTION Interlock_R10 : BOOL
VAR_INPUT
    signals : ARRAY[16] OF BOOL;
END_VAR
    Interlock_R10 := signals[10] AND signals[0];
END_FUNCTION
FUNCTION Interlock_R11 : BOOL
VAR_INPUT
    signals : ARRAY[16] OF BOOL;
END_VAR
    Interlock_R11 := signals[11] AND signals[0];
END_FUNCTION
FUNCTION Interlock_R12 : BOOL
VAR_INPUT
    signals : ARRAY[16] OF BOOL;
END_VAR
    Interlock_R12 := signals[12] AND signals[0];
END_FUNCTION
FUNCTION Interlock_R13 : BOOL
VAR_INPUT
    signals : ARRAY[16] OF BOOL;
END_VAR
    Interlock_R13 := signals[13] AND signals[0];
END_FUNCTION
FUNCTION Interlock_R14 : BOOL
VAR_INPUT
    signals : ARRAY[16] OF BOOL;
END_VAR
    Interlock_R14 := signals[14] AND signals[0];
END_FUNCTION
FUNCTION Interlock_R15 : BOOL
VAR_INPUT
    signals : ARRAY[16] OF BOOL;
END_VAR
    Interlock_R15 := signals[15] AND signals[0];
END_FUNCTION
(* ================================================================ *)
(* 报警管理系统 *)
(* ================================================================ *)

FUNCTION AlarmManager : INT
VAR_INPUT
    alarm_signals : ARRAY[16] OF BOOL;
END_VAR
VAR
    alm_idx : INT;
    active_count : INT;
END_VAR
    active_count := 0;
    FOR alm_idx := 0 TO 15 DO
        IF alarm_signals[alm_idx] THEN
            active_count := active_count + 1;
        END_IF;
    END_FOR;
    AlarmManager := active_count;
END_FUNCTION

FUNCTION Alarm_P1_A0 : BOOL
VAR_INPUT
    trigger : BOOL;
END_VAR
    alarm_counter := alarm_counter + 1;
    Alarm_P1_A0 := trigger;
END_FUNCTION
FUNCTION Alarm_P1_A1 : BOOL
VAR_INPUT
    trigger : BOOL;
END_VAR
    alarm_counter := alarm_counter + 1;
    Alarm_P1_A1 := trigger;
END_FUNCTION
FUNCTION Alarm_P1_A2 : BOOL
VAR_INPUT
    trigger : BOOL;
END_VAR
    alarm_counter := alarm_counter + 1;
    Alarm_P1_A2 := trigger;
END_FUNCTION
FUNCTION Alarm_P1_A3 : BOOL
VAR_INPUT
    trigger : BOOL;
END_VAR
    alarm_counter := alarm_counter + 1;
    Alarm_P1_A3 := trigger;
END_FUNCTION
FUNCTION Alarm_P2_A0 : BOOL
VAR_INPUT
    trigger : BOOL;
END_VAR
    alarm_counter := alarm_counter + 1;
    Alarm_P2_A0 := trigger;
END_FUNCTION
FUNCTION Alarm_P2_A1 : BOOL
VAR_INPUT
    trigger : BOOL;
END_VAR
    alarm_counter := alarm_counter + 1;
    Alarm_P2_A1 := trigger;
END_FUNCTION
FUNCTION Alarm_P2_A2 : BOOL
VAR_INPUT
    trigger : BOOL;
END_VAR
    alarm_counter := alarm_counter + 1;
    Alarm_P2_A2 := trigger;
END_FUNCTION
FUNCTION Alarm_P2_A3 : BOOL
VAR_INPUT
    trigger : BOOL;
END_VAR
    alarm_counter := alarm_counter + 1;
    Alarm_P2_A3 := trigger;
END_FUNCTION
FUNCTION Alarm_P3_A0 : BOOL
VAR_INPUT
    trigger : BOOL;
END_VAR
    alarm_counter := alarm_counter + 1;
    Alarm_P3_A0 := trigger;
END_FUNCTION
FUNCTION Alarm_P3_A1 : BOOL
VAR_INPUT
    trigger : BOOL;
END_VAR
    alarm_counter := alarm_counter + 1;
    Alarm_P3_A1 := trigger;
END_FUNCTION
FUNCTION Alarm_P3_A2 : BOOL
VAR_INPUT
    trigger : BOOL;
END_VAR
    alarm_counter := alarm_counter + 1;
    Alarm_P3_A2 := trigger;
END_FUNCTION
FUNCTION Alarm_P3_A3 : BOOL
VAR_INPUT
    trigger : BOOL;
END_VAR
    alarm_counter := alarm_counter + 1;
    Alarm_P3_A3 := trigger;
END_FUNCTION
FUNCTION Alarm_P4_A0 : BOOL
VAR_INPUT
    trigger : BOOL;
END_VAR
    alarm_counter := alarm_counter + 1;
    Alarm_P4_A0 := trigger;
END_FUNCTION
FUNCTION Alarm_P4_A1 : BOOL
VAR_INPUT
    trigger : BOOL;
END_VAR
    alarm_counter := alarm_counter + 1;
    Alarm_P4_A1 := trigger;
END_FUNCTION
FUNCTION Alarm_P4_A2 : BOOL
VAR_INPUT
    trigger : BOOL;
END_VAR
    alarm_counter := alarm_counter + 1;
    Alarm_P4_A2 := trigger;
END_FUNCTION
FUNCTION Alarm_P4_A3 : BOOL
VAR_INPUT
    trigger : BOOL;
END_VAR
    alarm_counter := alarm_counter + 1;
    Alarm_P4_A3 := trigger;
END_FUNCTION
(* ================================================================ *)
(* 反应堆状态机 *)
(* ================================================================ *)

FUNCTION StateMachine : INT
VAR_INPUT
    trip : BOOL;
END_VAR
VAR
    next_state : INT;
END_VAR
    next_state := system_state;
    IF trip THEN
        next_state := SYS_EMERGENCY;
    ELSIF system_state = SYS_IDLE THEN
        next_state := SYS_STARTUP;
    ELSIF system_state = SYS_STARTUP THEN
        next_state := SYS_RUNNING;
    ELSIF system_state = SYS_RUNNING THEN
        next_state := SYS_RUNNING;
    ELSIF system_state = SYS_EMERGENCY THEN
        next_state := SYS_SHUTDOWN;
    ELSIF system_state = SYS_SHUTDOWN THEN
        next_state := SYS_IDLE;
    END_IF;
    StateMachine := next_state;
END_FUNCTION

(* ================================================================ *)
(* 主控制周期 - 包含所有子系统 *)
(* ================================================================ *)

FUNCTION ControlCycle
VAR
    s0 : QREAL;
    s1 : QREAL;
    s2 : QREAL;
    s3 : QREAL;
    s4 : QREAL;
    s5 : QREAL;
    s6 : QREAL;
    s7 : QREAL;
    trip_cond : BOOL;
    avg_temp : REAL;
    avg_press : REAL;
    pid_temp : REAL;
    pid_press : REAL;
    pid_flow : REAL;
    pid_level : REAL;
    alm_signals : ARRAY[16] OF BOOL;
    alm_idx : INT;
    alm_cnt : INT;
END_VAR

    (* 读取所有传感器 *)
    s0 := SensorGroup0_Vote();
    s1 := SensorGroup1_Vote();
    s2 := SensorGroup2_Vote();
    s3 := SensorGroup3_Vote();
    s4 := SensorGroup4_Vote();
    s5 := SensorGroup5_Vote();
    s6 := SensorGroup6_Vote();
    s7 := SensorGroup7_Vote();

    (* 质量检查 *)
    tmp_int := GetQuality(s0);
    IF tmp_int > 1 THEN fault_counter := fault_counter + 1; END_IF;

    (* 2oo4 表决汇总 *)
    avg_temp := (ToReal(s0) + ToReal(s1) + ToReal(s2) + ToReal(s3)) / 4.0;
    avg_press := (ToReal(s4) + ToReal(s5) + ToReal(s6) + ToReal(s7)) / 4.0;

    (* PID 计算 *)
    pid_temp := PID_Temperature(500.0, avg_temp);
    pid_press := PID_Pressure(10.0, avg_press);
    pid_flow := PID_Flow(200.0, avg_temp * 0.5);
    pid_level := PID_Level(5.0, avg_press * 0.3);

    (* 跳闸判断 *)
    trip_cond := FALSE;
    IF avg_temp > TEMP_TRIP THEN trip_cond := TRUE; END_IF;
    IF avg_press > PRESS_TRIP THEN trip_cond := TRUE; END_IF;
    IF trip_cond THEN trip_counter := trip_counter + 1; END_IF;

    (* 报警更新 *)
    FOR alm_idx := 0 TO 15 DO
        alm_signals[alm_idx] := FALSE;
    END_FOR;
    IF avg_temp > TEMP_TRIP THEN alm_signals[0] := TRUE; END_IF;
    IF avg_press > PRESS_TRIP THEN alm_signals[1] := TRUE; END_IF;
    alm_cnt := AlarmManager(alm_signals);
    alarm_counter := alarm_counter + alm_cnt;

    (* 状态机 *)
    system_state := StateMachine(trip_cond);

    scan_counter := scan_counter + 1;
END_FUNCTION

(* @LOOP_MAX(100) - 校验函数 1 *)
FUNCTION Verify_Channel_1 : INT
VAR_INPUT
    value : REAL;
    limit : REAL;
END_VAR
    tmp_bool := (value <= limit);
    IF tmp_bool THEN
        Verify_Channel_1 := 0;
    ELSE
        Verify_Channel_1 := -1;
    END_IF;
END_FUNCTION

FUNCTION Scale_1 : REAL
VAR_INPUT
    raw : REAL;
END_VAR
    tmp_real := raw * 1.1;
    IF tmp_real > 10000.0 THEN
        tmp_real := 10000.0;
    END_IF;
    Scale_1 := tmp_real;
END_FUNCTION

FUNCTION LimitCheck_1 : BOOL
VAR_INPUT
    value : REAL;
    lo : REAL;
    hi : REAL;
END_VAR
    LimitCheck_1 := (value >= lo) AND (value <= hi);
END_FUNCTION

(* @LOOP_MAX(100) - 校验函数 2 *)
FUNCTION Verify_Channel_2 : INT
VAR_INPUT
    value : REAL;
    limit : REAL;
END_VAR
    tmp_bool := (value <= limit);
    IF tmp_bool THEN
        Verify_Channel_2 := 0;
    ELSE
        Verify_Channel_2 := -1;
    END_IF;
END_FUNCTION

FUNCTION Scale_2 : REAL
VAR_INPUT
    raw : REAL;
END_VAR
    tmp_real := raw * 1.2;
    IF tmp_real > 10000.0 THEN
        tmp_real := 10000.0;
    END_IF;
    Scale_2 := tmp_real;
END_FUNCTION

FUNCTION LimitCheck_2 : BOOL
VAR_INPUT
    value : REAL;
    lo : REAL;
    hi : REAL;
END_VAR
    LimitCheck_2 := (value >= lo) AND (value <= hi);
END_FUNCTION

(* @LOOP_MAX(100) - 校验函数 3 *)
FUNCTION Verify_Channel_3 : INT
VAR_INPUT
    value : REAL;
    limit : REAL;
END_VAR
    tmp_bool := (value <= limit);
    IF tmp_bool THEN
        Verify_Channel_3 := 0;
    ELSE
        Verify_Channel_3 := -1;
    END_IF;
END_FUNCTION

FUNCTION Scale_3 : REAL
VAR_INPUT
    raw : REAL;
END_VAR
    tmp_real := raw * 1.3;
    IF tmp_real > 10000.0 THEN
        tmp_real := 10000.0;
    END_IF;
    Scale_3 := tmp_real;
END_FUNCTION

FUNCTION LimitCheck_3 : BOOL
VAR_INPUT
    value : REAL;
    lo : REAL;
    hi : REAL;
END_VAR
    LimitCheck_3 := (value >= lo) AND (value <= hi);
END_FUNCTION

(* @LOOP_MAX(100) - 校验函数 4 *)
FUNCTION Verify_Channel_4 : INT
VAR_INPUT
    value : REAL;
    limit : REAL;
END_VAR
    tmp_bool := (value <= limit);
    IF tmp_bool THEN
        Verify_Channel_4 := 0;
    ELSE
        Verify_Channel_4 := -1;
    END_IF;
END_FUNCTION

FUNCTION Scale_4 : REAL
VAR_INPUT
    raw : REAL;
END_VAR
    tmp_real := raw * 1.4;
    IF tmp_real > 10000.0 THEN
        tmp_real := 10000.0;
    END_IF;
    Scale_4 := tmp_real;
END_FUNCTION

FUNCTION LimitCheck_4 : BOOL
VAR_INPUT
    value : REAL;
    lo : REAL;
    hi : REAL;
END_VAR
    LimitCheck_4 := (value >= lo) AND (value <= hi);
END_FUNCTION

(* @LOOP_MAX(100) - 校验函数 5 *)
FUNCTION Verify_Channel_5 : INT
VAR_INPUT
    value : REAL;
    limit : REAL;
END_VAR
    tmp_bool := (value <= limit);
    IF tmp_bool THEN
        Verify_Channel_5 := 0;
    ELSE
        Verify_Channel_5 := -1;
    END_IF;
END_FUNCTION

FUNCTION Scale_5 : REAL
VAR_INPUT
    raw : REAL;
END_VAR
    tmp_real := raw * 1.5;
    IF tmp_real > 10000.0 THEN
        tmp_real := 10000.0;
    END_IF;
    Scale_5 := tmp_real;
END_FUNCTION

FUNCTION LimitCheck_5 : BOOL
VAR_INPUT
    value : REAL;
    lo : REAL;
    hi : REAL;
END_VAR
    LimitCheck_5 := (value >= lo) AND (value <= hi);
END_FUNCTION

(* @LOOP_MAX(100) - 校验函数 6 *)
FUNCTION Verify_Channel_6 : INT
VAR_INPUT
    value : REAL;
    limit : REAL;
END_VAR
    tmp_bool := (value <= limit);
    IF tmp_bool THEN
        Verify_Channel_6 := 0;
    ELSE
        Verify_Channel_6 := -1;
    END_IF;
END_FUNCTION

FUNCTION Scale_6 : REAL
VAR_INPUT
    raw : REAL;
END_VAR
    tmp_real := raw * 1.6;
    IF tmp_real > 10000.0 THEN
        tmp_real := 10000.0;
    END_IF;
    Scale_6 := tmp_real;
END_FUNCTION

FUNCTION LimitCheck_6 : BOOL
VAR_INPUT
    value : REAL;
    lo : REAL;
    hi : REAL;
END_VAR
    LimitCheck_6 := (value >= lo) AND (value <= hi);
END_FUNCTION

(* @LOOP_MAX(100) - 校验函数 7 *)
FUNCTION Verify_Channel_7 : INT
VAR_INPUT
    value : REAL;
    limit : REAL;
END_VAR
    tmp_bool := (value <= limit);
    IF tmp_bool THEN
        Verify_Channel_7 := 0;
    ELSE
        Verify_Channel_7 := -1;
    END_IF;
END_FUNCTION

FUNCTION Scale_7 : REAL
VAR_INPUT
    raw : REAL;
END_VAR
    tmp_real := raw * 1.7;
    IF tmp_real > 10000.0 THEN
        tmp_real := 10000.0;
    END_IF;
    Scale_7 := tmp_real;
END_FUNCTION

FUNCTION LimitCheck_7 : BOOL
VAR_INPUT
    value : REAL;
    lo : REAL;
    hi : REAL;
END_VAR
    LimitCheck_7 := (value >= lo) AND (value <= hi);
END_FUNCTION

(* @LOOP_MAX(100) - 校验函数 8 *)
FUNCTION Verify_Channel_8 : INT
VAR_INPUT
    value : REAL;
    limit : REAL;
END_VAR
    tmp_bool := (value <= limit);
    IF tmp_bool THEN
        Verify_Channel_8 := 0;
    ELSE
        Verify_Channel_8 := -1;
    END_IF;
END_FUNCTION

FUNCTION Scale_8 : REAL
VAR_INPUT
    raw : REAL;
END_VAR
    tmp_real := raw * 1.8;
    IF tmp_real > 10000.0 THEN
        tmp_real := 10000.0;
    END_IF;
    Scale_8 := tmp_real;
END_FUNCTION

FUNCTION LimitCheck_8 : BOOL
VAR_INPUT
    value : REAL;
    lo : REAL;
    hi : REAL;
END_VAR
    LimitCheck_8 := (value >= lo) AND (value <= hi);
END_FUNCTION

(* @LOOP_MAX(100) - 校验函数 9 *)
FUNCTION Verify_Channel_9 : INT
VAR_INPUT
    value : REAL;
    limit : REAL;
END_VAR
    tmp_bool := (value <= limit);
    IF tmp_bool THEN
        Verify_Channel_9 := 0;
    ELSE
        Verify_Channel_9 := -1;
    END_IF;
END_FUNCTION

FUNCTION Scale_9 : REAL
VAR_INPUT
    raw : REAL;
END_VAR
    tmp_real := raw * 1.9;
    IF tmp_real > 10000.0 THEN
        tmp_real := 10000.0;
    END_IF;
    Scale_9 := tmp_real;
END_FUNCTION

FUNCTION LimitCheck_9 : BOOL
VAR_INPUT
    value : REAL;
    lo : REAL;
    hi : REAL;
END_VAR
    LimitCheck_9 := (value >= lo) AND (value <= hi);
END_FUNCTION

(* @LOOP_MAX(100) - 校验函数 10 *)
FUNCTION Verify_Channel_10 : INT
VAR_INPUT
    value : REAL;
    limit : REAL;
END_VAR
    tmp_bool := (value <= limit);
    IF tmp_bool THEN
        Verify_Channel_10 := 0;
    ELSE
        Verify_Channel_10 := -1;
    END_IF;
END_FUNCTION

FUNCTION Scale_10 : REAL
VAR_INPUT
    raw : REAL;
END_VAR
    tmp_real := raw * 1.10;
    IF tmp_real > 10000.0 THEN
        tmp_real := 10000.0;
    END_IF;
    Scale_10 := tmp_real;
END_FUNCTION

FUNCTION LimitCheck_10 : BOOL
VAR_INPUT
    value : REAL;
    lo : REAL;
    hi : REAL;
END_VAR
    LimitCheck_10 := (value >= lo) AND (value <= hi);
END_FUNCTION

(* @LOOP_MAX(100) - 校验函数 11 *)
FUNCTION Verify_Channel_11 : INT
VAR_INPUT
    value : REAL;
    limit : REAL;
END_VAR
    tmp_bool := (value <= limit);
    IF tmp_bool THEN
        Verify_Channel_11 := 0;
    ELSE
        Verify_Channel_11 := -1;
    END_IF;
END_FUNCTION

FUNCTION Scale_11 : REAL
VAR_INPUT
    raw : REAL;
END_VAR
    tmp_real := raw * 1.11;
    IF tmp_real > 10000.0 THEN
        tmp_real := 10000.0;
    END_IF;
    Scale_11 := tmp_real;
END_FUNCTION

FUNCTION LimitCheck_11 : BOOL
VAR_INPUT
    value : REAL;
    lo : REAL;
    hi : REAL;
END_VAR
    LimitCheck_11 := (value >= lo) AND (value <= hi);
END_FUNCTION

(* @LOOP_MAX(100) - 校验函数 12 *)
FUNCTION Verify_Channel_12 : INT
VAR_INPUT
    value : REAL;
    limit : REAL;
END_VAR
    tmp_bool := (value <= limit);
    IF tmp_bool THEN
        Verify_Channel_12 := 0;
    ELSE
        Verify_Channel_12 := -1;
    END_IF;
END_FUNCTION

FUNCTION Scale_12 : REAL
VAR_INPUT
    raw : REAL;
END_VAR
    tmp_real := raw * 1.12;
    IF tmp_real > 10000.0 THEN
        tmp_real := 10000.0;
    END_IF;
    Scale_12 := tmp_real;
END_FUNCTION

FUNCTION LimitCheck_12 : BOOL
VAR_INPUT
    value : REAL;
    lo : REAL;
    hi : REAL;
END_VAR
    LimitCheck_12 := (value >= lo) AND (value <= hi);
END_FUNCTION

(* @LOOP_MAX(100) - 校验函数 13 *)
FUNCTION Verify_Channel_13 : INT
VAR_INPUT
    value : REAL;
    limit : REAL;
END_VAR
    tmp_bool := (value <= limit);
    IF tmp_bool THEN
        Verify_Channel_13 := 0;
    ELSE
        Verify_Channel_13 := -1;
    END_IF;
END_FUNCTION

FUNCTION Scale_13 : REAL
VAR_INPUT
    raw : REAL;
END_VAR
    tmp_real := raw * 1.13;
    IF tmp_real > 10000.0 THEN
        tmp_real := 10000.0;
    END_IF;
    Scale_13 := tmp_real;
END_FUNCTION

FUNCTION LimitCheck_13 : BOOL
VAR_INPUT
    value : REAL;
    lo : REAL;
    hi : REAL;
END_VAR
    LimitCheck_13 := (value >= lo) AND (value <= hi);
END_FUNCTION

(* @LOOP_MAX(100) - 校验函数 14 *)
FUNCTION Verify_Channel_14 : INT
VAR_INPUT
    value : REAL;
    limit : REAL;
END_VAR
    tmp_bool := (value <= limit);
    IF tmp_bool THEN
        Verify_Channel_14 := 0;
    ELSE
        Verify_Channel_14 := -1;
    END_IF;
END_FUNCTION

FUNCTION Scale_14 : REAL
VAR_INPUT
    raw : REAL;
END_VAR
    tmp_real := raw * 1.14;
    IF tmp_real > 10000.0 THEN
        tmp_real := 10000.0;
    END_IF;
    Scale_14 := tmp_real;
END_FUNCTION

FUNCTION LimitCheck_14 : BOOL
VAR_INPUT
    value : REAL;
    lo : REAL;
    hi : REAL;
END_VAR
    LimitCheck_14 := (value >= lo) AND (value <= hi);
END_FUNCTION

(* @LOOP_MAX(100) - 校验函数 15 *)
FUNCTION Verify_Channel_15 : INT
VAR_INPUT
    value : REAL;
    limit : REAL;
END_VAR
    tmp_bool := (value <= limit);
    IF tmp_bool THEN
        Verify_Channel_15 := 0;
    ELSE
        Verify_Channel_15 := -1;
    END_IF;
END_FUNCTION

FUNCTION Scale_15 : REAL
VAR_INPUT
    raw : REAL;
END_VAR
    tmp_real := raw * 1.15;
    IF tmp_real > 10000.0 THEN
        tmp_real := 10000.0;
    END_IF;
    Scale_15 := tmp_real;
END_FUNCTION

FUNCTION LimitCheck_15 : BOOL
VAR_INPUT
    value : REAL;
    lo : REAL;
    hi : REAL;
END_VAR
    LimitCheck_15 := (value >= lo) AND (value <= hi);
END_FUNCTION

(* @LOOP_MAX(100) - 校验函数 16 *)
FUNCTION Verify_Channel_16 : INT
VAR_INPUT
    value : REAL;
    limit : REAL;
END_VAR
    tmp_bool := (value <= limit);
    IF tmp_bool THEN
        Verify_Channel_16 := 0;
    ELSE
        Verify_Channel_16 := -1;
    END_IF;
END_FUNCTION

FUNCTION Scale_16 : REAL
VAR_INPUT
    raw : REAL;
END_VAR
    tmp_real := raw * 1.16;
    IF tmp_real > 10000.0 THEN
        tmp_real := 10000.0;
    END_IF;
    Scale_16 := tmp_real;
END_FUNCTION

FUNCTION LimitCheck_16 : BOOL
VAR_INPUT
    value : REAL;
    lo : REAL;
    hi : REAL;
END_VAR
    LimitCheck_16 := (value >= lo) AND (value <= hi);
END_FUNCTION

(* @LOOP_MAX(100) - 校验函数 17 *)
FUNCTION Verify_Channel_17 : INT
VAR_INPUT
    value : REAL;
    limit : REAL;
END_VAR
    tmp_bool := (value <= limit);
    IF tmp_bool THEN
        Verify_Channel_17 := 0;
    ELSE
        Verify_Channel_17 := -1;
    END_IF;
END_FUNCTION

FUNCTION Scale_17 : REAL
VAR_INPUT
    raw : REAL;
END_VAR
    tmp_real := raw * 1.17;
    IF tmp_real > 10000.0 THEN
        tmp_real := 10000.0;
    END_IF;
    Scale_17 := tmp_real;
END_FUNCTION

FUNCTION LimitCheck_17 : BOOL
VAR_INPUT
    value : REAL;
    lo : REAL;
    hi : REAL;
END_VAR
    LimitCheck_17 := (value >= lo) AND (value <= hi);
END_FUNCTION

(* @LOOP_MAX(100) - 校验函数 18 *)
FUNCTION Verify_Channel_18 : INT
VAR_INPUT
    value : REAL;
    limit : REAL;
END_VAR
    tmp_bool := (value <= limit);
    IF tmp_bool THEN
        Verify_Channel_18 := 0;
    ELSE
        Verify_Channel_18 := -1;
    END_IF;
END_FUNCTION

FUNCTION Scale_18 : REAL
VAR_INPUT
    raw : REAL;
END_VAR
    tmp_real := raw * 1.18;
    IF tmp_real > 10000.0 THEN
        tmp_real := 10000.0;
    END_IF;
    Scale_18 := tmp_real;
END_FUNCTION

FUNCTION LimitCheck_18 : BOOL
VAR_INPUT
    value : REAL;
    lo : REAL;
    hi : REAL;
END_VAR
    LimitCheck_18 := (value >= lo) AND (value <= hi);
END_FUNCTION

(* @LOOP_MAX(100) - 校验函数 19 *)
FUNCTION Verify_Channel_19 : INT
VAR_INPUT
    value : REAL;
    limit : REAL;
END_VAR
    tmp_bool := (value <= limit);
    IF tmp_bool THEN
        Verify_Channel_19 := 0;
    ELSE
        Verify_Channel_19 := -1;
    END_IF;
END_FUNCTION

FUNCTION Scale_19 : REAL
VAR_INPUT
    raw : REAL;
END_VAR
    tmp_real := raw * 1.19;
    IF tmp_real > 10000.0 THEN
        tmp_real := 10000.0;
    END_IF;
    Scale_19 := tmp_real;
END_FUNCTION

FUNCTION LimitCheck_19 : BOOL
VAR_INPUT
    value : REAL;
    lo : REAL;
    hi : REAL;
END_VAR
    LimitCheck_19 := (value >= lo) AND (value <= hi);
END_FUNCTION

(* @LOOP_MAX(100) - 校验函数 20 *)
FUNCTION Verify_Channel_20 : INT
VAR_INPUT
    value : REAL;
    limit : REAL;
END_VAR
    tmp_bool := (value <= limit);
    IF tmp_bool THEN
        Verify_Channel_20 := 0;
    ELSE
        Verify_Channel_20 := -1;
    END_IF;
END_FUNCTION

FUNCTION Scale_20 : REAL
VAR_INPUT
    raw : REAL;
END_VAR
    tmp_real := raw * 1.20;
    IF tmp_real > 10000.0 THEN
        tmp_real := 10000.0;
    END_IF;
    Scale_20 := tmp_real;
END_FUNCTION

FUNCTION LimitCheck_20 : BOOL
VAR_INPUT
    value : REAL;
    lo : REAL;
    hi : REAL;
END_VAR
    LimitCheck_20 := (value >= lo) AND (value <= hi);
END_FUNCTION

(* @LOOP_MAX(100) - 校验函数 21 *)
FUNCTION Verify_Channel_21 : INT
VAR_INPUT
    value : REAL;
    limit : REAL;
END_VAR
    tmp_bool := (value <= limit);
    IF tmp_bool THEN
        Verify_Channel_21 := 0;
    ELSE
        Verify_Channel_21 := -1;
    END_IF;
END_FUNCTION

FUNCTION Scale_21 : REAL
VAR_INPUT
    raw : REAL;
END_VAR
    tmp_real := raw * 1.21;
    IF tmp_real > 10000.0 THEN
        tmp_real := 10000.0;
    END_IF;
    Scale_21 := tmp_real;
END_FUNCTION

FUNCTION LimitCheck_21 : BOOL
VAR_INPUT
    value : REAL;
    lo : REAL;
    hi : REAL;
END_VAR
    LimitCheck_21 := (value >= lo) AND (value <= hi);
END_FUNCTION

(* @LOOP_MAX(100) - 校验函数 22 *)
FUNCTION Verify_Channel_22 : INT
VAR_INPUT
    value : REAL;
    limit : REAL;
END_VAR
    tmp_bool := (value <= limit);
    IF tmp_bool THEN
        Verify_Channel_22 := 0;
    ELSE
        Verify_Channel_22 := -1;
    END_IF;
END_FUNCTION

FUNCTION Scale_22 : REAL
VAR_INPUT
    raw : REAL;
END_VAR
    tmp_real := raw * 1.22;
    IF tmp_real > 10000.0 THEN
        tmp_real := 10000.0;
    END_IF;
    Scale_22 := tmp_real;
END_FUNCTION

FUNCTION LimitCheck_22 : BOOL
VAR_INPUT
    value : REAL;
    lo : REAL;
    hi : REAL;
END_VAR
    LimitCheck_22 := (value >= lo) AND (value <= hi);
END_FUNCTION

(* @LOOP_MAX(100) - 校验函数 23 *)
FUNCTION Verify_Channel_23 : INT
VAR_INPUT
    value : REAL;
    limit : REAL;
END_VAR
    tmp_bool := (value <= limit);
    IF tmp_bool THEN
        Verify_Channel_23 := 0;
    ELSE
        Verify_Channel_23 := -1;
    END_IF;
END_FUNCTION

FUNCTION Scale_23 : REAL
VAR_INPUT
    raw : REAL;
END_VAR
    tmp_real := raw * 1.23;
    IF tmp_real > 10000.0 THEN
        tmp_real := 10000.0;
    END_IF;
    Scale_23 := tmp_real;
END_FUNCTION

FUNCTION LimitCheck_23 : BOOL
VAR_INPUT
    value : REAL;
    lo : REAL;
    hi : REAL;
END_VAR
    LimitCheck_23 := (value >= lo) AND (value <= hi);
END_FUNCTION

(* @LOOP_MAX(100) - 校验函数 24 *)
FUNCTION Verify_Channel_24 : INT
VAR_INPUT
    value : REAL;
    limit : REAL;
END_VAR
    tmp_bool := (value <= limit);
    IF tmp_bool THEN
        Verify_Channel_24 := 0;
    ELSE
        Verify_Channel_24 := -1;
    END_IF;
END_FUNCTION

FUNCTION Scale_24 : REAL
VAR_INPUT
    raw : REAL;
END_VAR
    tmp_real := raw * 1.24;
    IF tmp_real > 10000.0 THEN
        tmp_real := 10000.0;
    END_IF;
    Scale_24 := tmp_real;
END_FUNCTION

FUNCTION LimitCheck_24 : BOOL
VAR_INPUT
    value : REAL;
    lo : REAL;
    hi : REAL;
END_VAR
    LimitCheck_24 := (value >= lo) AND (value <= hi);
END_FUNCTION

(* @LOOP_MAX(100) - 校验函数 25 *)
FUNCTION Verify_Channel_25 : INT
VAR_INPUT
    value : REAL;
    limit : REAL;
END_VAR
    tmp_bool := (value <= limit);
    IF tmp_bool THEN
        Verify_Channel_25 := 0;
    ELSE
        Verify_Channel_25 := -1;
    END_IF;
END_FUNCTION

FUNCTION Scale_25 : REAL
VAR_INPUT
    raw : REAL;
END_VAR
    tmp_real := raw * 1.25;
    IF tmp_real > 10000.0 THEN
        tmp_real := 10000.0;
    END_IF;
    Scale_25 := tmp_real;
END_FUNCTION

FUNCTION LimitCheck_25 : BOOL
VAR_INPUT
    value : REAL;
    lo : REAL;
    hi : REAL;
END_VAR
    LimitCheck_25 := (value >= lo) AND (value <= hi);
END_FUNCTION

(* @LOOP_MAX(100) - 校验函数 26 *)
FUNCTION Verify_Channel_26 : INT
VAR_INPUT
    value : REAL;
    limit : REAL;
END_VAR
    tmp_bool := (value <= limit);
    IF tmp_bool THEN
        Verify_Channel_26 := 0;
    ELSE
        Verify_Channel_26 := -1;
    END_IF;
END_FUNCTION

FUNCTION Scale_26 : REAL
VAR_INPUT
    raw : REAL;
END_VAR
    tmp_real := raw * 1.26;
    IF tmp_real > 10000.0 THEN
        tmp_real := 10000.0;
    END_IF;
    Scale_26 := tmp_real;
END_FUNCTION

FUNCTION LimitCheck_26 : BOOL
VAR_INPUT
    value : REAL;
    lo : REAL;
    hi : REAL;
END_VAR
    LimitCheck_26 := (value >= lo) AND (value <= hi);
END_FUNCTION

(* @LOOP_MAX(100) - 校验函数 27 *)
FUNCTION Verify_Channel_27 : INT
VAR_INPUT
    value : REAL;
    limit : REAL;
END_VAR
    tmp_bool := (value <= limit);
    IF tmp_bool THEN
        Verify_Channel_27 := 0;
    ELSE
        Verify_Channel_27 := -1;
    END_IF;
END_FUNCTION

FUNCTION Scale_27 : REAL
VAR_INPUT
    raw : REAL;
END_VAR
    tmp_real := raw * 1.27;
    IF tmp_real > 10000.0 THEN
        tmp_real := 10000.0;
    END_IF;
    Scale_27 := tmp_real;
END_FUNCTION

FUNCTION LimitCheck_27 : BOOL
VAR_INPUT
    value : REAL;
    lo : REAL;
    hi : REAL;
END_VAR
    LimitCheck_27 := (value >= lo) AND (value <= hi);
END_FUNCTION

(* @LOOP_MAX(100) - 校验函数 28 *)
FUNCTION Verify_Channel_28 : INT
VAR_INPUT
    value : REAL;
    limit : REAL;
END_VAR
    tmp_bool := (value <= limit);
    IF tmp_bool THEN
        Verify_Channel_28 := 0;
    ELSE
        Verify_Channel_28 := -1;
    END_IF;
END_FUNCTION

FUNCTION Scale_28 : REAL
VAR_INPUT
    raw : REAL;
END_VAR
    tmp_real := raw * 1.28;
    IF tmp_real > 10000.0 THEN
        tmp_real := 10000.0;
    END_IF;
    Scale_28 := tmp_real;
END_FUNCTION

FUNCTION LimitCheck_28 : BOOL
VAR_INPUT
    value : REAL;
    lo : REAL;
    hi : REAL;
END_VAR
    LimitCheck_28 := (value >= lo) AND (value <= hi);
END_FUNCTION

(* @LOOP_MAX(100) - 校验函数 29 *)
FUNCTION Verify_Channel_29 : INT
VAR_INPUT
    value : REAL;
    limit : REAL;
END_VAR
    tmp_bool := (value <= limit);
    IF tmp_bool THEN
        Verify_Channel_29 := 0;
    ELSE
        Verify_Channel_29 := -1;
    END_IF;
END_FUNCTION

FUNCTION Scale_29 : REAL
VAR_INPUT
    raw : REAL;
END_VAR
    tmp_real := raw * 1.29;
    IF tmp_real > 10000.0 THEN
        tmp_real := 10000.0;
    END_IF;
    Scale_29 := tmp_real;
END_FUNCTION

FUNCTION LimitCheck_29 : BOOL
VAR_INPUT
    value : REAL;
    lo : REAL;
    hi : REAL;
END_VAR
    LimitCheck_29 := (value >= lo) AND (value <= hi);
END_FUNCTION

(* @LOOP_MAX(100) - 校验函数 30 *)
FUNCTION Verify_Channel_30 : INT
VAR_INPUT
    value : REAL;
    limit : REAL;
END_VAR
    tmp_bool := (value <= limit);
    IF tmp_bool THEN
        Verify_Channel_30 := 0;
    ELSE
        Verify_Channel_30 := -1;
    END_IF;
END_FUNCTION

FUNCTION Scale_30 : REAL
VAR_INPUT
    raw : REAL;
END_VAR
    tmp_real := raw * 1.30;
    IF tmp_real > 10000.0 THEN
        tmp_real := 10000.0;
    END_IF;
    Scale_30 := tmp_real;
END_FUNCTION

FUNCTION LimitCheck_30 : BOOL
VAR_INPUT
    value : REAL;
    lo : REAL;
    hi : REAL;
END_VAR
    LimitCheck_30 := (value >= lo) AND (value <= hi);
END_FUNCTION

(* @LOOP_MAX(100) - 校验函数 31 *)
FUNCTION Verify_Channel_31 : INT
VAR_INPUT
    value : REAL;
    limit : REAL;
END_VAR
    tmp_bool := (value <= limit);
    IF tmp_bool THEN
        Verify_Channel_31 := 0;
    ELSE
        Verify_Channel_31 := -1;
    END_IF;
END_FUNCTION

FUNCTION Scale_31 : REAL
VAR_INPUT
    raw : REAL;
END_VAR
    tmp_real := raw * 1.31;
    IF tmp_real > 10000.0 THEN
        tmp_real := 10000.0;
    END_IF;
    Scale_31 := tmp_real;
END_FUNCTION

FUNCTION LimitCheck_31 : BOOL
VAR_INPUT
    value : REAL;
    lo : REAL;
    hi : REAL;
END_VAR
    LimitCheck_31 := (value >= lo) AND (value <= hi);
END_FUNCTION

(* @LOOP_MAX(100) - 校验函数 32 *)
FUNCTION Verify_Channel_32 : INT
VAR_INPUT
    value : REAL;
    limit : REAL;
END_VAR
    tmp_bool := (value <= limit);
    IF tmp_bool THEN
        Verify_Channel_32 := 0;
    ELSE
        Verify_Channel_32 := -1;
    END_IF;
END_FUNCTION

FUNCTION Scale_32 : REAL
VAR_INPUT
    raw : REAL;
END_VAR
    tmp_real := raw * 1.32;
    IF tmp_real > 10000.0 THEN
        tmp_real := 10000.0;
    END_IF;
    Scale_32 := tmp_real;
END_FUNCTION

FUNCTION LimitCheck_32 : BOOL
VAR_INPUT
    value : REAL;
    lo : REAL;
    hi : REAL;
END_VAR
    LimitCheck_32 := (value >= lo) AND (value <= hi);
END_FUNCTION

(* @LOOP_MAX(100) - 校验函数 33 *)
FUNCTION Verify_Channel_33 : INT
VAR_INPUT
    value : REAL;
    limit : REAL;
END_VAR
    tmp_bool := (value <= limit);
    IF tmp_bool THEN
        Verify_Channel_33 := 0;
    ELSE
        Verify_Channel_33 := -1;
    END_IF;
END_FUNCTION

FUNCTION Scale_33 : REAL
VAR_INPUT
    raw : REAL;
END_VAR
    tmp_real := raw * 1.33;
    IF tmp_real > 10000.0 THEN
        tmp_real := 10000.0;
    END_IF;
    Scale_33 := tmp_real;
END_FUNCTION

FUNCTION LimitCheck_33 : BOOL
VAR_INPUT
    value : REAL;
    lo : REAL;
    hi : REAL;
END_VAR
    LimitCheck_33 := (value >= lo) AND (value <= hi);
END_FUNCTION

(* @LOOP_MAX(100) - 校验函数 34 *)
FUNCTION Verify_Channel_34 : INT
VAR_INPUT
    value : REAL;
    limit : REAL;
END_VAR
    tmp_bool := (value <= limit);
    IF tmp_bool THEN
        Verify_Channel_34 := 0;
    ELSE
        Verify_Channel_34 := -1;
    END_IF;
END_FUNCTION

FUNCTION Scale_34 : REAL
VAR_INPUT
    raw : REAL;
END_VAR
    tmp_real := raw * 1.34;
    IF tmp_real > 10000.0 THEN
        tmp_real := 10000.0;
    END_IF;
    Scale_34 := tmp_real;
END_FUNCTION

FUNCTION LimitCheck_34 : BOOL
VAR_INPUT
    value : REAL;
    lo : REAL;
    hi : REAL;
END_VAR
    LimitCheck_34 := (value >= lo) AND (value <= hi);
END_FUNCTION

(* @LOOP_MAX(100) - 校验函数 35 *)
FUNCTION Verify_Channel_35 : INT
VAR_INPUT
    value : REAL;
    limit : REAL;
END_VAR
    tmp_bool := (value <= limit);
    IF tmp_bool THEN
        Verify_Channel_35 := 0;
    ELSE
        Verify_Channel_35 := -1;
    END_IF;
END_FUNCTION

FUNCTION Scale_35 : REAL
VAR_INPUT
    raw : REAL;
END_VAR
    tmp_real := raw * 1.35;
    IF tmp_real > 10000.0 THEN
        tmp_real := 10000.0;
    END_IF;
    Scale_35 := tmp_real;
END_FUNCTION

FUNCTION LimitCheck_35 : BOOL
VAR_INPUT
    value : REAL;
    lo : REAL;
    hi : REAL;
END_VAR
    LimitCheck_35 := (value >= lo) AND (value <= hi);
END_FUNCTION

(* @LOOP_MAX(100) - 校验函数 36 *)
FUNCTION Verify_Channel_36 : INT
VAR_INPUT
    value : REAL;
    limit : REAL;
END_VAR
    tmp_bool := (value <= limit);
    IF tmp_bool THEN
        Verify_Channel_36 := 0;
    ELSE
        Verify_Channel_36 := -1;
    END_IF;
END_FUNCTION

FUNCTION Scale_36 : REAL
VAR_INPUT
    raw : REAL;
END_VAR
    tmp_real := raw * 1.36;
    IF tmp_real > 10000.0 THEN
        tmp_real := 10000.0;
    END_IF;
    Scale_36 := tmp_real;
END_FUNCTION

FUNCTION LimitCheck_36 : BOOL
VAR_INPUT
    value : REAL;
    lo : REAL;
    hi : REAL;
END_VAR
    LimitCheck_36 := (value >= lo) AND (value <= hi);
END_FUNCTION

(* @LOOP_MAX(100) - 校验函数 37 *)
FUNCTION Verify_Channel_37 : INT
VAR_INPUT
    value : REAL;
    limit : REAL;
END_VAR
    tmp_bool := (value <= limit);
    IF tmp_bool THEN
        Verify_Channel_37 := 0;
    ELSE
        Verify_Channel_37 := -1;
    END_IF;
END_FUNCTION

FUNCTION Scale_37 : REAL
VAR_INPUT
    raw : REAL;
END_VAR
    tmp_real := raw * 1.37;
    IF tmp_real > 10000.0 THEN
        tmp_real := 10000.0;
    END_IF;
    Scale_37 := tmp_real;
END_FUNCTION

FUNCTION LimitCheck_37 : BOOL
VAR_INPUT
    value : REAL;
    lo : REAL;
    hi : REAL;
END_VAR
    LimitCheck_37 := (value >= lo) AND (value <= hi);
END_FUNCTION

(* @LOOP_MAX(100) - 校验函数 38 *)
FUNCTION Verify_Channel_38 : INT
VAR_INPUT
    value : REAL;
    limit : REAL;
END_VAR
    tmp_bool := (value <= limit);
    IF tmp_bool THEN
        Verify_Channel_38 := 0;
    ELSE
        Verify_Channel_38 := -1;
    END_IF;
END_FUNCTION

FUNCTION Scale_38 : REAL
VAR_INPUT
    raw : REAL;
END_VAR
    tmp_real := raw * 1.38;
    IF tmp_real > 10000.0 THEN
        tmp_real := 10000.0;
    END_IF;
    Scale_38 := tmp_real;
END_FUNCTION

FUNCTION LimitCheck_38 : BOOL
VAR_INPUT
    value : REAL;
    lo : REAL;
    hi : REAL;
END_VAR
    LimitCheck_38 := (value >= lo) AND (value <= hi);
END_FUNCTION

(* @LOOP_MAX(100) - 校验函数 39 *)
FUNCTION Verify_Channel_39 : INT
VAR_INPUT
    value : REAL;
    limit : REAL;
END_VAR
    tmp_bool := (value <= limit);
    IF tmp_bool THEN
        Verify_Channel_39 := 0;
    ELSE
        Verify_Channel_39 := -1;
    END_IF;
END_FUNCTION

FUNCTION Scale_39 : REAL
VAR_INPUT
    raw : REAL;
END_VAR
    tmp_real := raw * 1.39;
    IF tmp_real > 10000.0 THEN
        tmp_real := 10000.0;
    END_IF;
    Scale_39 := tmp_real;
END_FUNCTION

FUNCTION LimitCheck_39 : BOOL
VAR_INPUT
    value : REAL;
    lo : REAL;
    hi : REAL;
END_VAR
    LimitCheck_39 := (value >= lo) AND (value <= hi);
END_FUNCTION

(* @LOOP_MAX(100) - 校验函数 40 *)
FUNCTION Verify_Channel_40 : INT
VAR_INPUT
    value : REAL;
    limit : REAL;
END_VAR
    tmp_bool := (value <= limit);
    IF tmp_bool THEN
        Verify_Channel_40 := 0;
    ELSE
        Verify_Channel_40 := -1;
    END_IF;
END_FUNCTION

FUNCTION Scale_40 : REAL
VAR_INPUT
    raw : REAL;
END_VAR
    tmp_real := raw * 1.40;
    IF tmp_real > 10000.0 THEN
        tmp_real := 10000.0;
    END_IF;
    Scale_40 := tmp_real;
END_FUNCTION

FUNCTION LimitCheck_40 : BOOL
VAR_INPUT
    value : REAL;
    lo : REAL;
    hi : REAL;
END_VAR
    LimitCheck_40 := (value >= lo) AND (value <= hi);
END_FUNCTION

(* @LOOP_MAX(100) - 校验函数 41 *)
FUNCTION Verify_Channel_41 : INT
VAR_INPUT
    value : REAL;
    limit : REAL;
END_VAR
    tmp_bool := (value <= limit);
    IF tmp_bool THEN
        Verify_Channel_41 := 0;
    ELSE
        Verify_Channel_41 := -1;
    END_IF;
END_FUNCTION

FUNCTION Scale_41 : REAL
VAR_INPUT
    raw : REAL;
END_VAR
    tmp_real := raw * 1.41;
    IF tmp_real > 10000.0 THEN
        tmp_real := 10000.0;
    END_IF;
    Scale_41 := tmp_real;
END_FUNCTION

FUNCTION LimitCheck_41 : BOOL
VAR_INPUT
    value : REAL;
    lo : REAL;
    hi : REAL;
END_VAR
    LimitCheck_41 := (value >= lo) AND (value <= hi);
END_FUNCTION

(* @LOOP_MAX(100) - 校验函数 42 *)
FUNCTION Verify_Channel_42 : INT
VAR_INPUT
    value : REAL;
    limit : REAL;
END_VAR
    tmp_bool := (value <= limit);
    IF tmp_bool THEN
        Verify_Channel_42 := 0;
    ELSE
        Verify_Channel_42 := -1;
    END_IF;
END_FUNCTION

FUNCTION Scale_42 : REAL
VAR_INPUT
    raw : REAL;
END_VAR
    tmp_real := raw * 1.42;
    IF tmp_real > 10000.0 THEN
        tmp_real := 10000.0;
    END_IF;
    Scale_42 := tmp_real;
END_FUNCTION

FUNCTION LimitCheck_42 : BOOL
VAR_INPUT
    value : REAL;
    lo : REAL;
    hi : REAL;
END_VAR
    LimitCheck_42 := (value >= lo) AND (value <= hi);
END_FUNCTION

(* @LOOP_MAX(100) - 校验函数 43 *)
FUNCTION Verify_Channel_43 : INT
VAR_INPUT
    value : REAL;
    limit : REAL;
END_VAR
    tmp_bool := (value <= limit);
    IF tmp_bool THEN
        Verify_Channel_43 := 0;
    ELSE
        Verify_Channel_43 := -1;
    END_IF;
END_FUNCTION

FUNCTION Scale_43 : REAL
VAR_INPUT
    raw : REAL;
END_VAR
    tmp_real := raw * 1.43;
    IF tmp_real > 10000.0 THEN
        tmp_real := 10000.0;
    END_IF;
    Scale_43 := tmp_real;
END_FUNCTION

FUNCTION LimitCheck_43 : BOOL
VAR_INPUT
    value : REAL;
    lo : REAL;
    hi : REAL;
END_VAR
    LimitCheck_43 := (value >= lo) AND (value <= hi);
END_FUNCTION

(* @LOOP_MAX(100) - 校验函数 44 *)
FUNCTION Verify_Channel_44 : INT
VAR_INPUT
    value : REAL;
    limit : REAL;
END_VAR
    tmp_bool := (value <= limit);
    IF tmp_bool THEN
        Verify_Channel_44 := 0;
    ELSE
        Verify_Channel_44 := -1;
    END_IF;
END_FUNCTION

FUNCTION Scale_44 : REAL
VAR_INPUT
    raw : REAL;
END_VAR
    tmp_real := raw * 1.44;
    IF tmp_real > 10000.0 THEN
        tmp_real := 10000.0;
    END_IF;
    Scale_44 := tmp_real;
END_FUNCTION

FUNCTION LimitCheck_44 : BOOL
VAR_INPUT
    value : REAL;
    lo : REAL;
    hi : REAL;
END_VAR
    LimitCheck_44 := (value >= lo) AND (value <= hi);
END_FUNCTION

(* @LOOP_MAX(100) - 校验函数 45 *)
FUNCTION Verify_Channel_45 : INT
VAR_INPUT
    value : REAL;
    limit : REAL;
END_VAR
    tmp_bool := (value <= limit);
    IF tmp_bool THEN
        Verify_Channel_45 := 0;
    ELSE
        Verify_Channel_45 := -1;
    END_IF;
END_FUNCTION

FUNCTION Scale_45 : REAL
VAR_INPUT
    raw : REAL;
END_VAR
    tmp_real := raw * 1.45;
    IF tmp_real > 10000.0 THEN
        tmp_real := 10000.0;
    END_IF;
    Scale_45 := tmp_real;
END_FUNCTION

FUNCTION LimitCheck_45 : BOOL
VAR_INPUT
    value : REAL;
    lo : REAL;
    hi : REAL;
END_VAR
    LimitCheck_45 := (value >= lo) AND (value <= hi);
END_FUNCTION

(* @LOOP_MAX(100) - 校验函数 46 *)
FUNCTION Verify_Channel_46 : INT
VAR_INPUT
    value : REAL;
    limit : REAL;
END_VAR
    tmp_bool := (value <= limit);
    IF tmp_bool THEN
        Verify_Channel_46 := 0;
    ELSE
        Verify_Channel_46 := -1;
    END_IF;
END_FUNCTION

FUNCTION Scale_46 : REAL
VAR_INPUT
    raw : REAL;
END_VAR
    tmp_real := raw * 1.46;
    IF tmp_real > 10000.0 THEN
        tmp_real := 10000.0;
    END_IF;
    Scale_46 := tmp_real;
END_FUNCTION

FUNCTION LimitCheck_46 : BOOL
VAR_INPUT
    value : REAL;
    lo : REAL;
    hi : REAL;
END_VAR
    LimitCheck_46 := (value >= lo) AND (value <= hi);
END_FUNCTION

(* @LOOP_MAX(100) - 校验函数 47 *)
FUNCTION Verify_Channel_47 : INT
VAR_INPUT
    value : REAL;
    limit : REAL;
END_VAR
    tmp_bool := (value <= limit);
    IF tmp_bool THEN
        Verify_Channel_47 := 0;
    ELSE
        Verify_Channel_47 := -1;
    END_IF;
END_FUNCTION

FUNCTION Scale_47 : REAL
VAR_INPUT
    raw : REAL;
END_VAR
    tmp_real := raw * 1.47;
    IF tmp_real > 10000.0 THEN
        tmp_real := 10000.0;
    END_IF;
    Scale_47 := tmp_real;
END_FUNCTION

FUNCTION LimitCheck_47 : BOOL
VAR_INPUT
    value : REAL;
    lo : REAL;
    hi : REAL;
END_VAR
    LimitCheck_47 := (value >= lo) AND (value <= hi);
END_FUNCTION

(* @LOOP_MAX(100) - 校验函数 48 *)
FUNCTION Verify_Channel_48 : INT
VAR_INPUT
    value : REAL;
    limit : REAL;
END_VAR
    tmp_bool := (value <= limit);
    IF tmp_bool THEN
        Verify_Channel_48 := 0;
    ELSE
        Verify_Channel_48 := -1;
    END_IF;
END_FUNCTION

FUNCTION Scale_48 : REAL
VAR_INPUT
    raw : REAL;
END_VAR
    tmp_real := raw * 1.48;
    IF tmp_real > 10000.0 THEN
        tmp_real := 10000.0;
    END_IF;
    Scale_48 := tmp_real;
END_FUNCTION

FUNCTION LimitCheck_48 : BOOL
VAR_INPUT
    value : REAL;
    lo : REAL;
    hi : REAL;
END_VAR
    LimitCheck_48 := (value >= lo) AND (value <= hi);
END_FUNCTION

(* @LOOP_MAX(100) - 校验函数 49 *)
FUNCTION Verify_Channel_49 : INT
VAR_INPUT
    value : REAL;
    limit : REAL;
END_VAR
    tmp_bool := (value <= limit);
    IF tmp_bool THEN
        Verify_Channel_49 := 0;
    ELSE
        Verify_Channel_49 := -1;
    END_IF;
END_FUNCTION

FUNCTION Scale_49 : REAL
VAR_INPUT
    raw : REAL;
END_VAR
    tmp_real := raw * 1.49;
    IF tmp_real > 10000.0 THEN
        tmp_real := 10000.0;
    END_IF;
    Scale_49 := tmp_real;
END_FUNCTION

FUNCTION LimitCheck_49 : BOOL
VAR_INPUT
    value : REAL;
    lo : REAL;
    hi : REAL;
END_VAR
    LimitCheck_49 := (value >= lo) AND (value <= hi);
END_FUNCTION

(* @LOOP_MAX(100) - 校验函数 50 *)
FUNCTION Verify_Channel_50 : INT
VAR_INPUT
    value : REAL;
    limit : REAL;
END_VAR
    tmp_bool := (value <= limit);
    IF tmp_bool THEN
        Verify_Channel_50 := 0;
    ELSE
        Verify_Channel_50 := -1;
    END_IF;
END_FUNCTION

FUNCTION Scale_50 : REAL
VAR_INPUT
    raw : REAL;
END_VAR
    tmp_real := raw * 1.50;
    IF tmp_real > 10000.0 THEN
        tmp_real := 10000.0;
    END_IF;
    Scale_50 := tmp_real;
END_FUNCTION

FUNCTION LimitCheck_50 : BOOL
VAR_INPUT
    value : REAL;
    lo : REAL;
    hi : REAL;
END_VAR
    LimitCheck_50 := (value >= lo) AND (value <= hi);
END_FUNCTION

(* @LOOP_MAX(100) - 校验函数 51 *)
FUNCTION Verify_Channel_51 : INT
VAR_INPUT
    value : REAL;
    limit : REAL;
END_VAR
    tmp_bool := (value <= limit);
    IF tmp_bool THEN
        Verify_Channel_51 := 0;
    ELSE
        Verify_Channel_51 := -1;
    END_IF;
END_FUNCTION

FUNCTION Scale_51 : REAL
VAR_INPUT
    raw : REAL;
END_VAR
    tmp_real := raw * 1.51;
    IF tmp_real > 10000.0 THEN
        tmp_real := 10000.0;
    END_IF;
    Scale_51 := tmp_real;
END_FUNCTION

FUNCTION LimitCheck_51 : BOOL
VAR_INPUT
    value : REAL;
    lo : REAL;
    hi : REAL;
END_VAR
    LimitCheck_51 := (value >= lo) AND (value <= hi);
END_FUNCTION

(* @LOOP_MAX(100) - 校验函数 52 *)
FUNCTION Verify_Channel_52 : INT
VAR_INPUT
    value : REAL;
    limit : REAL;
END_VAR
    tmp_bool := (value <= limit);
    IF tmp_bool THEN
        Verify_Channel_52 := 0;
    ELSE
        Verify_Channel_52 := -1;
    END_IF;
END_FUNCTION

FUNCTION Scale_52 : REAL
VAR_INPUT
    raw : REAL;
END_VAR
    tmp_real := raw * 1.52;
    IF tmp_real > 10000.0 THEN
        tmp_real := 10000.0;
    END_IF;
    Scale_52 := tmp_real;
END_FUNCTION

FUNCTION LimitCheck_52 : BOOL
VAR_INPUT
    value : REAL;
    lo : REAL;
    hi : REAL;
END_VAR
    LimitCheck_52 := (value >= lo) AND (value <= hi);
END_FUNCTION

(* @LOOP_MAX(100) - 校验函数 53 *)
FUNCTION Verify_Channel_53 : INT
VAR_INPUT
    value : REAL;
    limit : REAL;
END_VAR
    tmp_bool := (value <= limit);
    IF tmp_bool THEN
        Verify_Channel_53 := 0;
    ELSE
        Verify_Channel_53 := -1;
    END_IF;
END_FUNCTION

FUNCTION Scale_53 : REAL
VAR_INPUT
    raw : REAL;
END_VAR
    tmp_real := raw * 1.53;
    IF tmp_real > 10000.0 THEN
        tmp_real := 10000.0;
    END_IF;
    Scale_53 := tmp_real;
END_FUNCTION

FUNCTION LimitCheck_53 : BOOL
VAR_INPUT
    value : REAL;
    lo : REAL;
    hi : REAL;
END_VAR
    LimitCheck_53 := (value >= lo) AND (value <= hi);
END_FUNCTION

(* @LOOP_MAX(100) - 校验函数 54 *)
FUNCTION Verify_Channel_54 : INT
VAR_INPUT
    value : REAL;
    limit : REAL;
END_VAR
    tmp_bool := (value <= limit);
    IF tmp_bool THEN
        Verify_Channel_54 := 0;
    ELSE
        Verify_Channel_54 := -1;
    END_IF;
END_FUNCTION

FUNCTION Scale_54 : REAL
VAR_INPUT
    raw : REAL;
END_VAR
    tmp_real := raw * 1.54;
    IF tmp_real > 10000.0 THEN
        tmp_real := 10000.0;
    END_IF;
    Scale_54 := tmp_real;
END_FUNCTION

FUNCTION LimitCheck_54 : BOOL
VAR_INPUT
    value : REAL;
    lo : REAL;
    hi : REAL;
END_VAR
    LimitCheck_54 := (value >= lo) AND (value <= hi);
END_FUNCTION

(* @LOOP_MAX(100) - 校验函数 55 *)
FUNCTION Verify_Channel_55 : INT
VAR_INPUT
    value : REAL;
    limit : REAL;
END_VAR
    tmp_bool := (value <= limit);
    IF tmp_bool THEN
        Verify_Channel_55 := 0;
    ELSE
        Verify_Channel_55 := -1;
    END_IF;
END_FUNCTION

FUNCTION Scale_55 : REAL
VAR_INPUT
    raw : REAL;
END_VAR
    tmp_real := raw * 1.55;
    IF tmp_real > 10000.0 THEN
        tmp_real := 10000.0;
    END_IF;
    Scale_55 := tmp_real;
END_FUNCTION

FUNCTION LimitCheck_55 : BOOL
VAR_INPUT
    value : REAL;
    lo : REAL;
    hi : REAL;
END_VAR
    LimitCheck_55 := (value >= lo) AND (value <= hi);
END_FUNCTION

(* @LOOP_MAX(100) - 校验函数 56 *)
FUNCTION Verify_Channel_56 : INT
VAR_INPUT
    value : REAL;
    limit : REAL;
END_VAR
    tmp_bool := (value <= limit);
    IF tmp_bool THEN
        Verify_Channel_56 := 0;
    ELSE
        Verify_Channel_56 := -1;
    END_IF;
END_FUNCTION

FUNCTION Scale_56 : REAL
VAR_INPUT
    raw : REAL;
END_VAR
    tmp_real := raw * 1.56;
    IF tmp_real > 10000.0 THEN
        tmp_real := 10000.0;
    END_IF;
    Scale_56 := tmp_real;
END_FUNCTION

FUNCTION LimitCheck_56 : BOOL
VAR_INPUT
    value : REAL;
    lo : REAL;
    hi : REAL;
END_VAR
    LimitCheck_56 := (value >= lo) AND (value <= hi);
END_FUNCTION

(* @LOOP_MAX(100) - 校验函数 57 *)
FUNCTION Verify_Channel_57 : INT
VAR_INPUT
    value : REAL;
    limit : REAL;
END_VAR
    tmp_bool := (value <= limit);
    IF tmp_bool THEN
        Verify_Channel_57 := 0;
    ELSE
        Verify_Channel_57 := -1;
    END_IF;
END_FUNCTION

FUNCTION Scale_57 : REAL
VAR_INPUT
    raw : REAL;
END_VAR
    tmp_real := raw * 1.57;
    IF tmp_real > 10000.0 THEN
        tmp_real := 10000.0;
    END_IF;
    Scale_57 := tmp_real;
END_FUNCTION

FUNCTION LimitCheck_57 : BOOL
VAR_INPUT
    value : REAL;
    lo : REAL;
    hi : REAL;
END_VAR
    LimitCheck_57 := (value >= lo) AND (value <= hi);
END_FUNCTION

(* @LOOP_MAX(100) - 校验函数 58 *)
FUNCTION Verify_Channel_58 : INT
VAR_INPUT
    value : REAL;
    limit : REAL;
END_VAR
    tmp_bool := (value <= limit);
    IF tmp_bool THEN
        Verify_Channel_58 := 0;
    ELSE
        Verify_Channel_58 := -1;
    END_IF;
END_FUNCTION

FUNCTION Scale_58 : REAL
VAR_INPUT
    raw : REAL;
END_VAR
    tmp_real := raw * 1.58;
    IF tmp_real > 10000.0 THEN
        tmp_real := 10000.0;
    END_IF;
    Scale_58 := tmp_real;
END_FUNCTION

FUNCTION LimitCheck_58 : BOOL
VAR_INPUT
    value : REAL;
    lo : REAL;
    hi : REAL;
END_VAR
    LimitCheck_58 := (value >= lo) AND (value <= hi);
END_FUNCTION

(* @LOOP_MAX(100) - 校验函数 59 *)
FUNCTION Verify_Channel_59 : INT
VAR_INPUT
    value : REAL;
    limit : REAL;
END_VAR
    tmp_bool := (value <= limit);
    IF tmp_bool THEN
        Verify_Channel_59 := 0;
    ELSE
        Verify_Channel_59 := -1;
    END_IF;
END_FUNCTION

FUNCTION Scale_59 : REAL
VAR_INPUT
    raw : REAL;
END_VAR
    tmp_real := raw * 1.59;
    IF tmp_real > 10000.0 THEN
        tmp_real := 10000.0;
    END_IF;
    Scale_59 := tmp_real;
END_FUNCTION

FUNCTION LimitCheck_59 : BOOL
VAR_INPUT
    value : REAL;
    lo : REAL;
    hi : REAL;
END_VAR
    LimitCheck_59 := (value >= lo) AND (value <= hi);
END_FUNCTION

(* @LOOP_MAX(100) - 校验函数 60 *)
FUNCTION Verify_Channel_60 : INT
VAR_INPUT
    value : REAL;
    limit : REAL;
END_VAR
    tmp_bool := (value <= limit);
    IF tmp_bool THEN
        Verify_Channel_60 := 0;
    ELSE
        Verify_Channel_60 := -1;
    END_IF;
END_FUNCTION

FUNCTION Scale_60 : REAL
VAR_INPUT
    raw : REAL;
END_VAR
    tmp_real := raw * 1.60;
    IF tmp_real > 10000.0 THEN
        tmp_real := 10000.0;
    END_IF;
    Scale_60 := tmp_real;
END_FUNCTION

FUNCTION LimitCheck_60 : BOOL
VAR_INPUT
    value : REAL;
    lo : REAL;
    hi : REAL;
END_VAR
    LimitCheck_60 := (value >= lo) AND (value <= hi);
END_FUNCTION

(* @LOOP_MAX(100) - 校验函数 61 *)
FUNCTION Verify_Channel_61 : INT
VAR_INPUT
    value : REAL;
    limit : REAL;
END_VAR
    tmp_bool := (value <= limit);
    IF tmp_bool THEN
        Verify_Channel_61 := 0;
    ELSE
        Verify_Channel_61 := -1;
    END_IF;
END_FUNCTION

FUNCTION Scale_61 : REAL
VAR_INPUT
    raw : REAL;
END_VAR
    tmp_real := raw * 1.61;
    IF tmp_real > 10000.0 THEN
        tmp_real := 10000.0;
    END_IF;
    Scale_61 := tmp_real;
END_FUNCTION

FUNCTION LimitCheck_61 : BOOL
VAR_INPUT
    value : REAL;
    lo : REAL;
    hi : REAL;
END_VAR
    LimitCheck_61 := (value >= lo) AND (value <= hi);
END_FUNCTION

(* @LOOP_MAX(100) - 校验函数 62 *)
FUNCTION Verify_Channel_62 : INT
VAR_INPUT
    value : REAL;
    limit : REAL;
END_VAR
    tmp_bool := (value <= limit);
    IF tmp_bool THEN
        Verify_Channel_62 := 0;
    ELSE
        Verify_Channel_62 := -1;
    END_IF;
END_FUNCTION

FUNCTION Scale_62 : REAL
VAR_INPUT
    raw : REAL;
END_VAR
    tmp_real := raw * 1.62;
    IF tmp_real > 10000.0 THEN
        tmp_real := 10000.0;
    END_IF;
    Scale_62 := tmp_real;
END_FUNCTION

FUNCTION LimitCheck_62 : BOOL
VAR_INPUT
    value : REAL;
    lo : REAL;
    hi : REAL;
END_VAR
    LimitCheck_62 := (value >= lo) AND (value <= hi);
END_FUNCTION

(* @LOOP_MAX(100) - 校验函数 63 *)
FUNCTION Verify_Channel_63 : INT
VAR_INPUT
    value : REAL;
    limit : REAL;
END_VAR
    tmp_bool := (value <= limit);
    IF tmp_bool THEN
        Verify_Channel_63 := 0;
    ELSE
        Verify_Channel_63 := -1;
    END_IF;
END_FUNCTION

FUNCTION Scale_63 : REAL
VAR_INPUT
    raw : REAL;
END_VAR
    tmp_real := raw * 1.63;
    IF tmp_real > 10000.0 THEN
        tmp_real := 10000.0;
    END_IF;
    Scale_63 := tmp_real;
END_FUNCTION

FUNCTION LimitCheck_63 : BOOL
VAR_INPUT
    value : REAL;
    lo : REAL;
    hi : REAL;
END_VAR
    LimitCheck_63 := (value >= lo) AND (value <= hi);
END_FUNCTION

(* @LOOP_MAX(100) - 校验函数 64 *)
FUNCTION Verify_Channel_64 : INT
VAR_INPUT
    value : REAL;
    limit : REAL;
END_VAR
    tmp_bool := (value <= limit);
    IF tmp_bool THEN
        Verify_Channel_64 := 0;
    ELSE
        Verify_Channel_64 := -1;
    END_IF;
END_FUNCTION

FUNCTION Scale_64 : REAL
VAR_INPUT
    raw : REAL;
END_VAR
    tmp_real := raw * 1.64;
    IF tmp_real > 10000.0 THEN
        tmp_real := 10000.0;
    END_IF;
    Scale_64 := tmp_real;
END_FUNCTION

FUNCTION LimitCheck_64 : BOOL
VAR_INPUT
    value : REAL;
    lo : REAL;
    hi : REAL;
END_VAR
    LimitCheck_64 := (value >= lo) AND (value <= hi);
END_FUNCTION

(* @LOOP_MAX(100) - 校验函数 65 *)
FUNCTION Verify_Channel_65 : INT
VAR_INPUT
    value : REAL;
    limit : REAL;
END_VAR
    tmp_bool := (value <= limit);
    IF tmp_bool THEN
        Verify_Channel_65 := 0;
    ELSE
        Verify_Channel_65 := -1;
    END_IF;
END_FUNCTION

FUNCTION Scale_65 : REAL
VAR_INPUT
    raw : REAL;
END_VAR
    tmp_real := raw * 1.65;
    IF tmp_real > 10000.0 THEN
        tmp_real := 10000.0;
    END_IF;
    Scale_65 := tmp_real;
END_FUNCTION

FUNCTION LimitCheck_65 : BOOL
VAR_INPUT
    value : REAL;
    lo : REAL;
    hi : REAL;
END_VAR
    LimitCheck_65 := (value >= lo) AND (value <= hi);
END_FUNCTION

(* @LOOP_MAX(100) - 校验函数 66 *)
FUNCTION Verify_Channel_66 : INT
VAR_INPUT
    value : REAL;
    limit : REAL;
END_VAR
    tmp_bool := (value <= limit);
    IF tmp_bool THEN
        Verify_Channel_66 := 0;
    ELSE
        Verify_Channel_66 := -1;
    END_IF;
END_FUNCTION

FUNCTION Scale_66 : REAL
VAR_INPUT
    raw : REAL;
END_VAR
    tmp_real := raw * 1.66;
    IF tmp_real > 10000.0 THEN
        tmp_real := 10000.0;
    END_IF;
    Scale_66 := tmp_real;
END_FUNCTION

FUNCTION LimitCheck_66 : BOOL
VAR_INPUT
    value : REAL;
    lo : REAL;
    hi : REAL;
END_VAR
    LimitCheck_66 := (value >= lo) AND (value <= hi);
END_FUNCTION

(* @LOOP_MAX(100) - 校验函数 67 *)
FUNCTION Verify_Channel_67 : INT
VAR_INPUT
    value : REAL;
    limit : REAL;
END_VAR
    tmp_bool := (value <= limit);
    IF tmp_bool THEN
        Verify_Channel_67 := 0;
    ELSE
        Verify_Channel_67 := -1;
    END_IF;
END_FUNCTION

FUNCTION Scale_67 : REAL
VAR_INPUT
    raw : REAL;
END_VAR
    tmp_real := raw * 1.67;
    IF tmp_real > 10000.0 THEN
        tmp_real := 10000.0;
    END_IF;
    Scale_67 := tmp_real;
END_FUNCTION

FUNCTION LimitCheck_67 : BOOL
VAR_INPUT
    value : REAL;
    lo : REAL;
    hi : REAL;
END_VAR
    LimitCheck_67 := (value >= lo) AND (value <= hi);
END_FUNCTION

(* @LOOP_MAX(100) - 校验函数 68 *)
FUNCTION Verify_Channel_68 : INT
VAR_INPUT
    value : REAL;
    limit : REAL;
END_VAR
    tmp_bool := (value <= limit);
    IF tmp_bool THEN
        Verify_Channel_68 := 0;
    ELSE
        Verify_Channel_68 := -1;
    END_IF;
END_FUNCTION

FUNCTION Scale_68 : REAL
VAR_INPUT
    raw : REAL;
END_VAR
    tmp_real := raw * 1.68;
    IF tmp_real > 10000.0 THEN
        tmp_real := 10000.0;
    END_IF;
    Scale_68 := tmp_real;
END_FUNCTION

FUNCTION LimitCheck_68 : BOOL
VAR_INPUT
    value : REAL;
    lo : REAL;
    hi : REAL;
END_VAR
    LimitCheck_68 := (value >= lo) AND (value <= hi);
END_FUNCTION

(* @LOOP_MAX(100) - 校验函数 69 *)
FUNCTION Verify_Channel_69 : INT
VAR_INPUT
    value : REAL;
    limit : REAL;
END_VAR
    tmp_bool := (value <= limit);
    IF tmp_bool THEN
        Verify_Channel_69 := 0;
    ELSE
        Verify_Channel_69 := -1;
    END_IF;
END_FUNCTION

FUNCTION Scale_69 : REAL
VAR_INPUT
    raw : REAL;
END_VAR
    tmp_real := raw * 1.69;
    IF tmp_real > 10000.0 THEN
        tmp_real := 10000.0;
    END_IF;
    Scale_69 := tmp_real;
END_FUNCTION

FUNCTION LimitCheck_69 : BOOL
VAR_INPUT
    value : REAL;
    lo : REAL;
    hi : REAL;
END_VAR
    LimitCheck_69 := (value >= lo) AND (value <= hi);
END_FUNCTION

(* @LOOP_MAX(100) - 校验函数 70 *)
FUNCTION Verify_Channel_70 : INT
VAR_INPUT
    value : REAL;
    limit : REAL;
END_VAR
    tmp_bool := (value <= limit);
    IF tmp_bool THEN
        Verify_Channel_70 := 0;
    ELSE
        Verify_Channel_70 := -1;
    END_IF;
END_FUNCTION

FUNCTION Scale_70 : REAL
VAR_INPUT
    raw : REAL;
END_VAR
    tmp_real := raw * 1.70;
    IF tmp_real > 10000.0 THEN
        tmp_real := 10000.0;
    END_IF;
    Scale_70 := tmp_real;
END_FUNCTION

FUNCTION LimitCheck_70 : BOOL
VAR_INPUT
    value : REAL;
    lo : REAL;
    hi : REAL;
END_VAR
    LimitCheck_70 := (value >= lo) AND (value <= hi);
END_FUNCTION

(* @LOOP_MAX(100) - 校验函数 71 *)
FUNCTION Verify_Channel_71 : INT
VAR_INPUT
    value : REAL;
    limit : REAL;
END_VAR
    tmp_bool := (value <= limit);
    IF tmp_bool THEN
        Verify_Channel_71 := 0;
    ELSE
        Verify_Channel_71 := -1;
    END_IF;
END_FUNCTION

FUNCTION Scale_71 : REAL
VAR_INPUT
    raw : REAL;
END_VAR
    tmp_real := raw * 1.71;
    IF tmp_real > 10000.0 THEN
        tmp_real := 10000.0;
    END_IF;
    Scale_71 := tmp_real;
END_FUNCTION

FUNCTION LimitCheck_71 : BOOL
VAR_INPUT
    value : REAL;
    lo : REAL;
    hi : REAL;
END_VAR
    LimitCheck_71 := (value >= lo) AND (value <= hi);
END_FUNCTION

(* @LOOP_MAX(100) - 校验函数 72 *)
FUNCTION Verify_Channel_72 : INT
VAR_INPUT
    value : REAL;
    limit : REAL;
END_VAR
    tmp_bool := (value <= limit);
    IF tmp_bool THEN
        Verify_Channel_72 := 0;
    ELSE
        Verify_Channel_72 := -1;
    END_IF;
END_FUNCTION

FUNCTION Scale_72 : REAL
VAR_INPUT
    raw : REAL;
END_VAR
    tmp_real := raw * 1.72;
    IF tmp_real > 10000.0 THEN
        tmp_real := 10000.0;
    END_IF;
    Scale_72 := tmp_real;
END_FUNCTION

FUNCTION LimitCheck_72 : BOOL
VAR_INPUT
    value : REAL;
    lo : REAL;
    hi : REAL;
END_VAR
    LimitCheck_72 := (value >= lo) AND (value <= hi);
END_FUNCTION

(* @LOOP_MAX(100) - 校验函数 73 *)
FUNCTION Verify_Channel_73 : INT
VAR_INPUT
    value : REAL;
    limit : REAL;
END_VAR
    tmp_bool := (value <= limit);
    IF tmp_bool THEN
        Verify_Channel_73 := 0;
    ELSE
        Verify_Channel_73 := -1;
    END_IF;
END_FUNCTION

FUNCTION Scale_73 : REAL
VAR_INPUT
    raw : REAL;
END_VAR
    tmp_real := raw * 1.73;
    IF tmp_real > 10000.0 THEN
        tmp_real := 10000.0;
    END_IF;
    Scale_73 := tmp_real;
END_FUNCTION

FUNCTION LimitCheck_73 : BOOL
VAR_INPUT
    value : REAL;
    lo : REAL;
    hi : REAL;
END_VAR
    LimitCheck_73 := (value >= lo) AND (value <= hi);
END_FUNCTION

(* @LOOP_MAX(100) - 校验函数 74 *)
FUNCTION Verify_Channel_74 : INT
VAR_INPUT
    value : REAL;
    limit : REAL;
END_VAR
    tmp_bool := (value <= limit);
    IF tmp_bool THEN
        Verify_Channel_74 := 0;
    ELSE
        Verify_Channel_74 := -1;
    END_IF;
END_FUNCTION

FUNCTION Scale_74 : REAL
VAR_INPUT
    raw : REAL;
END_VAR
    tmp_real := raw * 1.74;
    IF tmp_real > 10000.0 THEN
        tmp_real := 10000.0;
    END_IF;
    Scale_74 := tmp_real;
END_FUNCTION

FUNCTION LimitCheck_74 : BOOL
VAR_INPUT
    value : REAL;
    lo : REAL;
    hi : REAL;
END_VAR
    LimitCheck_74 := (value >= lo) AND (value <= hi);
END_FUNCTION

(* @LOOP_MAX(100) - 校验函数 75 *)
FUNCTION Verify_Channel_75 : INT
VAR_INPUT
    value : REAL;
    limit : REAL;
END_VAR
    tmp_bool := (value <= limit);
    IF tmp_bool THEN
        Verify_Channel_75 := 0;
    ELSE
        Verify_Channel_75 := -1;
    END_IF;
END_FUNCTION

FUNCTION Scale_75 : REAL
VAR_INPUT
    raw : REAL;
END_VAR
    tmp_real := raw * 1.75;
    IF tmp_real > 10000.0 THEN
        tmp_real := 10000.0;
    END_IF;
    Scale_75 := tmp_real;
END_FUNCTION

FUNCTION LimitCheck_75 : BOOL
VAR_INPUT
    value : REAL;
    lo : REAL;
    hi : REAL;
END_VAR
    LimitCheck_75 := (value >= lo) AND (value <= hi);
END_FUNCTION

(* @LOOP_MAX(100) - 校验函数 76 *)
FUNCTION Verify_Channel_76 : INT
VAR_INPUT
    value : REAL;
    limit : REAL;
END_VAR
    tmp_bool := (value <= limit);
    IF tmp_bool THEN
        Verify_Channel_76 := 0;
    ELSE
        Verify_Channel_76 := -1;
    END_IF;
END_FUNCTION

FUNCTION Scale_76 : REAL
VAR_INPUT
    raw : REAL;
END_VAR
    tmp_real := raw * 1.76;
    IF tmp_real > 10000.0 THEN
        tmp_real := 10000.0;
    END_IF;
    Scale_76 := tmp_real;
END_FUNCTION

FUNCTION LimitCheck_76 : BOOL
VAR_INPUT
    value : REAL;
    lo : REAL;
    hi : REAL;
END_VAR
    LimitCheck_76 := (value >= lo) AND (value <= hi);
END_FUNCTION

(* @LOOP_MAX(100) - 校验函数 77 *)
FUNCTION Verify_Channel_77 : INT
VAR_INPUT
    value : REAL;
    limit : REAL;
END_VAR
    tmp_bool := (value <= limit);
    IF tmp_bool THEN
        Verify_Channel_77 := 0;
    ELSE
        Verify_Channel_77 := -1;
    END_IF;
END_FUNCTION

FUNCTION Scale_77 : REAL
VAR_INPUT
    raw : REAL;
END_VAR
    tmp_real := raw * 1.77;
    IF tmp_real > 10000.0 THEN
        tmp_real := 10000.0;
    END_IF;
    Scale_77 := tmp_real;
END_FUNCTION

FUNCTION LimitCheck_77 : BOOL
VAR_INPUT
    value : REAL;
    lo : REAL;
    hi : REAL;
END_VAR
    LimitCheck_77 := (value >= lo) AND (value <= hi);
END_FUNCTION

(* @LOOP_MAX(100) - 校验函数 78 *)
FUNCTION Verify_Channel_78 : INT
VAR_INPUT
    value : REAL;
    limit : REAL;
END_VAR
    tmp_bool := (value <= limit);
    IF tmp_bool THEN
        Verify_Channel_78 := 0;
    ELSE
        Verify_Channel_78 := -1;
    END_IF;
END_FUNCTION

FUNCTION Scale_78 : REAL
VAR_INPUT
    raw : REAL;
END_VAR
    tmp_real := raw * 1.78;
    IF tmp_real > 10000.0 THEN
        tmp_real := 10000.0;
    END_IF;
    Scale_78 := tmp_real;
END_FUNCTION

FUNCTION LimitCheck_78 : BOOL
VAR_INPUT
    value : REAL;
    lo : REAL;
    hi : REAL;
END_VAR
    LimitCheck_78 := (value >= lo) AND (value <= hi);
END_FUNCTION

(* @LOOP_MAX(100) - 校验函数 79 *)
FUNCTION Verify_Channel_79 : INT
VAR_INPUT
    value : REAL;
    limit : REAL;
END_VAR
    tmp_bool := (value <= limit);
    IF tmp_bool THEN
        Verify_Channel_79 := 0;
    ELSE
        Verify_Channel_79 := -1;
    END_IF;
END_FUNCTION

FUNCTION Scale_79 : REAL
VAR_INPUT
    raw : REAL;
END_VAR
    tmp_real := raw * 1.79;
    IF tmp_real > 10000.0 THEN
        tmp_real := 10000.0;
    END_IF;
    Scale_79 := tmp_real;
END_FUNCTION

FUNCTION LimitCheck_79 : BOOL
VAR_INPUT
    value : REAL;
    lo : REAL;
    hi : REAL;
END_VAR
    LimitCheck_79 := (value >= lo) AND (value <= hi);
END_FUNCTION

(* @LOOP_MAX(100) - 校验函数 80 *)
FUNCTION Verify_Channel_80 : INT
VAR_INPUT
    value : REAL;
    limit : REAL;
END_VAR
    tmp_bool := (value <= limit);
    IF tmp_bool THEN
        Verify_Channel_80 := 0;
    ELSE
        Verify_Channel_80 := -1;
    END_IF;
END_FUNCTION

FUNCTION Scale_80 : REAL
VAR_INPUT
    raw : REAL;
END_VAR
    tmp_real := raw * 1.80;
    IF tmp_real > 10000.0 THEN
        tmp_real := 10000.0;
    END_IF;
    Scale_80 := tmp_real;
END_FUNCTION

FUNCTION LimitCheck_80 : BOOL
VAR_INPUT
    value : REAL;
    lo : REAL;
    hi : REAL;
END_VAR
    LimitCheck_80 := (value >= lo) AND (value <= hi);
END_FUNCTION

(* @LOOP_MAX(100) - 校验函数 81 *)
FUNCTION Verify_Channel_81 : INT
VAR_INPUT
    value : REAL;
    limit : REAL;
END_VAR
    tmp_bool := (value <= limit);
    IF tmp_bool THEN
        Verify_Channel_81 := 0;
    ELSE
        Verify_Channel_81 := -1;
    END_IF;
END_FUNCTION

FUNCTION Scale_81 : REAL
VAR_INPUT
    raw : REAL;
END_VAR
    tmp_real := raw * 1.81;
    IF tmp_real > 10000.0 THEN
        tmp_real := 10000.0;
    END_IF;
    Scale_81 := tmp_real;
END_FUNCTION

FUNCTION LimitCheck_81 : BOOL
VAR_INPUT
    value : REAL;
    lo : REAL;
    hi : REAL;
END_VAR
    LimitCheck_81 := (value >= lo) AND (value <= hi);
END_FUNCTION

(* @LOOP_MAX(100) - 校验函数 82 *)
FUNCTION Verify_Channel_82 : INT
VAR_INPUT
    value : REAL;
    limit : REAL;
END_VAR
    tmp_bool := (value <= limit);
    IF tmp_bool THEN
        Verify_Channel_82 := 0;
    ELSE
        Verify_Channel_82 := -1;
    END_IF;
END_FUNCTION

FUNCTION Scale_82 : REAL
VAR_INPUT
    raw : REAL;
END_VAR
    tmp_real := raw * 1.82;
    IF tmp_real > 10000.0 THEN
        tmp_real := 10000.0;
    END_IF;
    Scale_82 := tmp_real;
END_FUNCTION

FUNCTION LimitCheck_82 : BOOL
VAR_INPUT
    value : REAL;
    lo : REAL;
    hi : REAL;
END_VAR
    LimitCheck_82 := (value >= lo) AND (value <= hi);
END_FUNCTION

(* @LOOP_MAX(100) - 校验函数 83 *)
FUNCTION Verify_Channel_83 : INT
VAR_INPUT
    value : REAL;
    limit : REAL;
END_VAR
    tmp_bool := (value <= limit);
    IF tmp_bool THEN
        Verify_Channel_83 := 0;
    ELSE
        Verify_Channel_83 := -1;
    END_IF;
END_FUNCTION

FUNCTION Scale_83 : REAL
VAR_INPUT
    raw : REAL;
END_VAR
    tmp_real := raw * 1.83;
    IF tmp_real > 10000.0 THEN
        tmp_real := 10000.0;
    END_IF;
    Scale_83 := tmp_real;
END_FUNCTION

FUNCTION LimitCheck_83 : BOOL
VAR_INPUT
    value : REAL;
    lo : REAL;
    hi : REAL;
END_VAR
    LimitCheck_83 := (value >= lo) AND (value <= hi);
END_FUNCTION

(* @LOOP_MAX(100) - 校验函数 84 *)
FUNCTION Verify_Channel_84 : INT
VAR_INPUT
    value : REAL;
    limit : REAL;
END_VAR
    tmp_bool := (value <= limit);
    IF tmp_bool THEN
        Verify_Channel_84 := 0;
    ELSE
        Verify_Channel_84 := -1;
    END_IF;
END_FUNCTION

FUNCTION Scale_84 : REAL
VAR_INPUT
    raw : REAL;
END_VAR
    tmp_real := raw * 1.84;
    IF tmp_real > 10000.0 THEN
        tmp_real := 10000.0;
    END_IF;
    Scale_84 := tmp_real;
END_FUNCTION

FUNCTION LimitCheck_84 : BOOL
VAR_INPUT
    value : REAL;
    lo : REAL;
    hi : REAL;
END_VAR
    LimitCheck_84 := (value >= lo) AND (value <= hi);
END_FUNCTION

(* @LOOP_MAX(100) - 校验函数 85 *)
FUNCTION Verify_Channel_85 : INT
VAR_INPUT
    value : REAL;
    limit : REAL;
END_VAR
    tmp_bool := (value <= limit);
    IF tmp_bool THEN
        Verify_Channel_85 := 0;
    ELSE
        Verify_Channel_85 := -1;
    END_IF;
END_FUNCTION
